(* IEC 61131-3 sources: fse/dataset/original (part 3) *)

(* ---- lb_claude_assisted_30195e188caf_0084.st ---- *)
TYPE
  LOGLEVEL : (CRITICAL, WARNING, INFO, DEBUG) := INFO;
END_TYPE

FUNCTION_BLOCK LOGGER
  VAR_INPUT
    TRIG : BOOL;
    MSG : STRING;
    LEVEL : LOGLEVEL := INFO;
  END_VAR
  VAR
    TRIG0 : BOOL;
  END_VAR

  IF TRIG AND NOT TRIG0 THEN
  {{
   LogMessage(GetFbVar(LEVEL),(char*)GetFbVar(MSG, .body),GetFbVar(MSG, .len));
  }}
  END_IF;
  TRIG0:=TRIG;
END_FUNCTION_BLOCK

FUNCTION_BLOCK python_eval
  VAR_INPUT
    TRIG : BOOL;
    CODE : STRING;
  END_VAR
  VAR_OUTPUT
    ACK : BOOL;
    RESULT : STRING;
  END_VAR
  VAR
    STATE : DWORD;
    BUFFER : STRING;
    PREBUFFER : STRING;
    TRIGM1 : BOOL;
    TRIGGED : BOOL;
  END_VAR

  {extern void __PythonEvalFB(int, PYTHON_EVAL*);__PythonEvalFB(0, data__);}
END_FUNCTION_BLOCK

FUNCTION_BLOCK python_poll
  VAR_INPUT
    TRIG : BOOL;
    CODE : STRING;
  END_VAR
  VAR_OUTPUT
    ACK : BOOL;
    RESULT : STRING;
  END_VAR
  VAR
    STATE : DWORD;
    BUFFER : STRING;
    PREBUFFER : STRING;
    TRIGM1 : BOOL;
    TRIGGED : BOOL;
  END_VAR

  {extern void __PythonEvalFB(int, PYTHON_EVAL*);__PythonEvalFB(1,(PYTHON_EVAL*)(void*)data__);}
END_FUNCTION_BLOCK

FUNCTION_BLOCK python_gear
  VAR_INPUT
    N : UINT;
    TRIG : BOOL;
    CODE : STRING;
  END_VAR
  VAR_OUTPUT
    ACK : BOOL;
    RESULT : STRING;
  END_VAR
  VAR
    py_eval : python_eval;
    COUNTER : UINT;
    _TMP_ADD10_OUT : UINT;
    _TMP_EQ13_OUT : BOOL;
    _TMP_SEL15_OUT : UINT;
    _TMP_AND7_OUT : BOOL;
  END_VAR

  _TMP_ADD10_OUT := ADD(COUNTER, 1);
  _TMP_EQ13_OUT := EQ(N, _TMP_ADD10_OUT);
  _TMP_SEL15_OUT := SEL(_TMP_EQ13_OUT, _TMP_ADD10_OUT, 0);
  COUNTER := _TMP_SEL15_OUT;
  _TMP_AND7_OUT := AND(_TMP_EQ13_OUT, TRIG);
  py_eval(TRIG := _TMP_AND7_OUT, CODE := CODE);
  ACK := py_eval.ACK;
  RESULT := py_eval.RESULT;
END_FUNCTION_BLOCK

PROGRAM plc2
  VAR
    ColorSensor_RED : INT;
    ColorSensor_GREEN : INT;
    ColorSensor_BLUE : INT;
    RangeSensor : REAL := 100.0;
    Pump : BOOL := FALSE;
    Doser_RED : BOOL := FALSE;
    Doser_BLUE : BOOL := FALSE;
  END_VAR
  VAR
    settleTime : TIME := TIME#5s;
    doseTime : TIME := TIME#1s;
    shutDown : BOOL := FALSE;
    treatmentComplete : BOOL := FALSE;
  END_VAR
  VAR
    stage : INT := 0;
    desiredDistanceFill : REAL := 60.0;
  END_VAR
  VAR
    minRed : INT := 20;
    doseTimer : TON;
    settleTimer : TON;
  END_VAR

  CASE stage OF
      0:  (*Filling stage: it will fill up to a certain amount that corresponds to a certain distance*)

          IF RangeSensor > desiredDistanceFill THEN
            Pump := TRUE;
          ELSE
            Pump := FALSE;
            stage := 1;
          END_IF;

     1:  (*Treatment stage*)

          IF ColorSensor_RED < minRed THEN (*Ensure minimum red value is inserted*)
            stage := 2;
            Doser_RED := TRUE;
            doseTimer(IN:= NOT doseTimer.Q, PT:= doseTime);

          ELSIF ColorSensor_RED > ColorSensor_BLUE  THEN (*Ensure blue quantity is > Red *)

              stage := 3;
              Doser_BLUE := TRUE;
              doseTimer(IN:= NOT doseTimer.Q, PT:= doseTime);

          ELSE  (*Treatment complete*)

            stage := 5;

          END_IF;

      2:  (*Red Dosing Stage*)

          IF doseTimer.Q THEN
            Doser_RED := FALSE;
            stage := 4;
            doseTimer(IN:= FALSE);
            settleTimer(IN:= NOT settleTimer.Q, PT:= settleTime); (*let the dose settle*)
          END_IF;

      3: (* Blue Dosing Stage*)

          IF doseTimer.Q THEN
            Doser_BLUE := FALSE;
            stage := 4;
            doseTimer(IN:= FALSE);
            settleTimer(IN:= NOT settleTimer.Q, PT:= settleTime); (*let the dose settle*)
          END_IF;

      4: (*Settling Stage for Dosage*)

          IF settleTimer.Q THEN
          stage := 1;
          settleTimer(IN:=FALSE);
          END_IF;

      5: (*Treatment Complete*)

        treatmentComplete := TRUE;

  END_CASE;
END_PROGRAM

CONFIGURATION Config0

  RESOURCE Res0 ON PLC
    TASK task0(INTERVAL := T#200ms,PRIORITY := 0);
    PROGRAM instance0 WITH task0 : plc2;
  END_RESOURCE
END_CONFIGURATION

(* ---- lb_claude_assisted_30f898e237c2_0134.st ---- *)
FUNCTION_BLOCK T_PLC_MS_block
	VAR_OUTPUT
		T_PLC_MS :	UDINT;
	END_VAR

	VAR_EXTERNAL
		PLC_TICKS_PER_SEC :	INT;
		PLC_SYS_TICK_CNT :	DINT;
	END_VAR

	VAR
		debug :	BOOL;(*Debug-Mode ON / OFF*)
		N :	INT;(*Debug-Faktor*)
		Offset :	UDINT;(*Debug-Offset*)
		temp :	DWORD := DWORD#1;(*Debug-Offset*)
		mode :	BOOL;(*modus*)
		faktor :	UDINT;(*Systemtakt-Faktor*)
		init :	BOOL;
		v_plc_ticks_per_sec :	UDINT;
		base :	UDINT := UDINT#1000;
	END_VAR

	IF init = FALSE THEN
		v_plc_ticks_per_sec := INT_TO_UDINT(PLC_TICKS_PER_SEC);
		IF v_plc_ticks_per_sec = UDINT#1024 THEN
			faktor := UDINT#1;
			mode := FALSE;
		ELSIF v_plc_ticks_per_sec > UDINT#0 THEN
			IF v_plc_ticks_per_sec <= base THEN
				faktor := base / v_plc_ticks_per_sec;
				mode := FALSE;
			ELSE
				faktor := v_plc_ticks_per_sec / base;
				mode := TRUE;
			END_IF;
		ELSE
			faktor := UDINT#1;
		END_IF;
		init := TRUE;
	END_IF;

	IF mode THEN
		T_PLC_MS := DINT_TO_UDINT(PLC_SYS_TICK_CNT) / faktor;
	ELSE
		T_PLC_MS := DINT_TO_UDINT(PLC_SYS_TICK_CNT) * faktor;
	END_IF;

	IF debug THEN
		T_PLC_MS := (DWORD_TO_UDINT(SHL(UDINT_TO_DWORD(T_PLC_MS),N) OR SHL(temp,N)) - UDINT#1) + Offset;
	END_IF;
END_FUNCTION_BLOCK

FUNCTION_BLOCK INTEGRATE

	VAR_INPUT
		E :	BOOL := TRUE;
		X :	REAL;
		K :	REAL := 1.0;
	END_VAR

	VAR_IN_OUT
		Y :	REAL;
	END_VAR

	VAR
		X_last :	REAL;
		init :	BOOL;
		T_PLC_MS :	T_PLC_MS_block;
		last :	UDINT;
		tx :	UDINT;
	END_VAR

	T_PLC_MS();
	tx:= T_PLC_MS.T_PLC_MS;

	IF NOT init THEN
		init := TRUE;
		X_last := X;
	ELSIF E THEN
		Y := (X + X_LAST) * 0.5E-3 * UDINT_TO_REAL(tx-last) * K + Y;
		X_last := X;
	END_IF;
	last := tx;

END_FUNCTION_BLOCK

FUNCTION_BLOCK FT_INT_Block

	VAR_INPUT
		IN :	REAL;
		K :	REAL := 1.0;
		RUN :	BOOL := TRUE;
		RST :	BOOL;
		OUT_MIN :	REAL := REAL#-1.0E-37;
		OUT_MAX :	REAL := REAL#1.0E37;
	END_VAR

	VAR_OUTPUT
		OUT :	REAL;
		LIM :	BOOL;
	END_VAR

	VAR
		INTEG :	INTEGRATE;
	END_VAR

	IF rst THEN
		out := 0.0;
	ELSE
		integ(X := IN, E := RUN, K := K, Y := out);
		out := integ.Y;
	END_IF;

	(* limit the outputs *)
	IF out >= OUT_MAX THEN
		out := out_max;
		LIM := TRUE;
	ELSIF out <= out_min THEN
		out := out_min;
		lim := TRUE;
	ELSE
		lim := FALSE;
	END_IF;

END_FUNCTION_BLOCK

FUNCTION_BLOCK FT_PIW

	VAR_INPUT
		IN :	REAL;
		KP :	REAL := 1.0;
		KI :	REAL := 1.0;
		LIM_L :	REAL := -1.0E38;
		LIM_H :	REAL := 1.0E38;
		RST :	BOOL := FALSE;
	END_VAR

	VAR_OUTPUT
		Y :	REAL;
		LIM :	BOOL;
	END_VAR

	VAR
		integ :	FT_INT_Block;
	END_VAR

	integ(IN := IN, K := KI, RUN := NOT LIM, RST := RST);

	(* set output value *)
	Y := KP * IN + integ.Out;

	(* check for limits *)
	IF Y < LIM_L THEN
		Y := LIM_L;
		LIM := TRUE;
	ELSIF Y > LIM_H THEN
		Y := LIM_H;
		LIM := TRUE;
	ELSE
		LIM := FALSE;
	END_IF;

END_FUNCTION_BLOCK

PROGRAM program0
	VAR
		IN :	REAL;
		KP :	REAL := 1.0;
		KI :	REAL := 1.0;
		LIM_L :	REAL := -1.0E38;
		LIM_H :	REAL := 1.0E38;
		RST :	BOOL := FALSE;

		Y :	REAL;
		LIM :	BOOL;

		func_block : FT_PIW;
	END_VAR
	func_block.IN := IN;
	func_block.KP := KP;
	func_block.KI := KI;
	func_block.LIM_L := LIM_L;
	func_block.LIM_H := LIM_H;
	func_block.RST := RST;
	func_block();
	Y := func_block.Y;
	LIM := func_block.LIM;
END_PROGRAM

CONFIGURATION Config0

	VAR_GLOBAL
		PLC_TICKS_PER_SEC :	INT;
		PLC_SYS_TICK_CNT :	DINT;
	END_VAR

	RESOURCE Res0 ON PLC
		TASK task0(INTERVAL := T#20ms,PRIORITY := 0);
		PROGRAM instance0 WITH task0 : program0;
	END_RESOURCE

END_CONFIGURATION

(* ---- lb_claude_assisted_33ab4d28fcd8_0080.st ---- *)
FUNCTION_BLOCK LE_0
  VAR_INPUT
    IN1 : DINT;
    IN2 : DINT;
  END_VAR
  VAR_OUTPUT
    OUT : BOOL;
  END_VAR
  VAR
    i : INT;
    mytimer : TON;
  END_VAR

  OUT:=FALSE;
  IF IN1<=IN2 then
    OUT:=TRUE;
  END_IF;
  mytimer(IN := TRUE, PT := t#8000ms);
  i:=0;
  IF mytimer.Q = TRUE then
     WHILE i<4 do
      OUT:=TRUE;
    End_WHILE;
  End_IF;
END_FUNCTION_BLOCK

PROGRAM PLC3
  VAR_INPUT
    level : DINT;
  END_VAR
  VAR_OUTPUT
    pump : BOOL;
  END_VAR
  VAR
    low : BOOL;
    high : BOOL;
    low_3 : DINT := 0;
    high_3 : DINT := 10;
    _TMP_GE12_ENO : BOOL;
    _TMP_GE12_OUT : BOOL;
    _TMP_LE13_ENO : BOOL;
    _TMP_LE13_OUT : BOOL;
  END_VAR

  _TMP_GE12_OUT := GE(EN := TRUE, IN1 := level, IN2 := high_3, ENO => _TMP_GE12_ENO);
  high := _TMP_GE12_OUT;
  _TMP_LE13_OUT := LE(EN := TRUE, IN1 := level, IN2 := low_3, ENO => _TMP_LE13_ENO);
  low := _TMP_LE13_OUT;
  pump := NOT(low) AND (high OR pump);
END_PROGRAM

PROGRAM PLC2
  VAR_INPUT
    level : DINT;
  END_VAR
  VAR_OUTPUT
    request : BOOL;
  END_VAR
  VAR
    open_req : BOOL;
    close_req : BOOL;
    low_2 : DINT := 10;
    high_2 : DINT := 20;
    LE_00 : LE_0;
    _TMP_GE11_ENO : BOOL;
    _TMP_GE11_OUT : BOOL;
  END_VAR

  _TMP_GE11_OUT := GE(EN := TRUE, IN1 := level, IN2 := high_2, ENO => _TMP_GE11_ENO);
  close_req := _TMP_GE11_OUT;
  LE_00(EN := TRUE, IN1 := level, IN2 := low_2);
  open_req := LE_00.OUT;
  request := NOT(close_req) AND (open_req OR request);
END_PROGRAM

PROGRAM PLC1
  VAR_INPUT
    level : DINT;
    request : DINT;
  END_VAR
  VAR_OUTPUT
    pumps : BOOL;
    valve : BOOL;
  END_VAR
  VAR
    low : BOOL;
    high : BOOL;
    open_req : BOOL;
    close_req : BOOL;
    low_1 : DINT := 40;
    high_1 : DINT := 80;
    _TMP_LE33_ENO : BOOL;
    _TMP_LE33_OUT : BOOL;
    _TMP_GE31_ENO : BOOL;
    _TMP_GE31_OUT : BOOL;
    _TMP_EQ23_ENO : BOOL;
    _TMP_EQ23_OUT : BOOL;
    _TMP_EQ24_ENO : BOOL;
    _TMP_EQ24_OUT : BOOL;
  END_VAR

  _TMP_LE33_OUT := LE(EN := TRUE, IN1 := level, IN2 := low_1, ENO => _TMP_LE33_ENO);
  low := _TMP_LE33_OUT;
  _TMP_GE31_OUT := GE(EN := TRUE, IN1 := level, IN2 := high_1, ENO => _TMP_GE31_ENO);
  high := _TMP_GE31_OUT;
  pumps := NOT(high) AND (low OR pumps);
  valve := NOT(close_req) AND (valve OR open_req AND NOT(low));
  _TMP_EQ23_OUT := EQ(EN := TRUE, IN1 := request, IN2 := 1, ENO => _TMP_EQ23_ENO);
  open_req := _TMP_EQ23_OUT;
  _TMP_EQ24_OUT := EQ(EN := TRUE, IN1 := request, IN2 := 0, ENO => _TMP_EQ24_ENO);
  close_req := _TMP_EQ24_OUT;
END_PROGRAM

CONFIGURATION Config0

  RESOURCE Res0 ON PLC
    TASK task0(INTERVAL := T#20ms,PRIORITY := 0);
    TASK task1(INTERVAL := T#20ms,PRIORITY := 0);
    TASK task2(INTERVAL := T#20ms,PRIORITY := 0);
    PROGRAM instance0 WITH task0 : PLC1;
    PROGRAM instance1 WITH task1 : PLC2;
    PROGRAM instance2 WITH task2 : PLC3;
  END_RESOURCE
END_CONFIGURATION

(* ---- lb_claude_assisted_33b79055e2cc_0056.st ---- *)
FUNCTION_BLOCK T_PLC_MS_block

	VAR_OUTPUT
		T_PLC_MS :	UDINT;
	END_VAR

	VAR_EXTERNAL
		PLC_TICKS_PER_SEC :	INT;
		PLC_SYS_TICK_CNT :	DINT;
	END_VAR

	VAR
		debug :	BOOL;(*Debug-Mode ON / OFF*)
		N :	INT;(*Debug-Faktor*)
		Offset :	UDINT;(*Debug-Offset*)
		temp :	DWORD := DWORD#1;(*Debug-Offset*)
		mode :	BOOL;(*modus*)
		faktor :	UDINT;(*Systemtakt-Faktor*)
		init :	BOOL;
		v_plc_ticks_per_sec :	UDINT;
		base :	UDINT := UDINT#1000;
	END_VAR

	IF init = FALSE THEN
		v_plc_ticks_per_sec := INT_TO_UDINT(PLC_TICKS_PER_SEC);
		IF v_plc_ticks_per_sec = UDINT#1024 THEN
			faktor := UDINT#1;
			mode := FALSE;
		ELSIF v_plc_ticks_per_sec > UDINT#0 THEN
			IF v_plc_ticks_per_sec <= base THEN
				faktor := base / v_plc_ticks_per_sec;
				mode := FALSE;
			ELSE
				faktor := v_plc_ticks_per_sec / base;
				mode := TRUE;
			END_IF;
		ELSE
			faktor := UDINT#1;
		END_IF;
		init := TRUE;
	END_IF;

	IF mode THEN
		T_PLC_MS := DINT_TO_UDINT(PLC_SYS_TICK_CNT) / faktor;
	ELSE
		T_PLC_MS := DINT_TO_UDINT(PLC_SYS_TICK_CNT) * faktor;
	END_IF;

	IF debug THEN
		T_PLC_MS := (DWORD_TO_UDINT(SHL(UDINT_TO_DWORD(T_PLC_MS),N) OR SHL(temp,N)) - UDINT#1) + Offset;
	END_IF;

END_FUNCTION_BLOCK

PROGRAM program0

	VAR
		LocalOUT  : UDINT;
		func_block : T_PLC_MS_block;
  	END_VAR

	func_block();
	LocalOUT := func_block.T_PLC_MS;

END_PROGRAM

CONFIGURATION Config0

	VAR_GLOBAL
		PLC_TICKS_PER_SEC :	INT;
		PLC_SYS_TICK_CNT :	DINT;
	END_VAR

  	RESOURCE Res0 ON PLC
    	TASK task0(INTERVAL := T#20ms,PRIORITY := 0);
    	PROGRAM instance0 WITH task0 : program0;
  	END_RESOURCE

END_CONFIGURATION

(* ---- lb_claude_assisted_350444d9c29e_0021.st ---- *)
(*
This code implements a randomly grown symbolic expression:

xor(xor(!((!(((xor(xor(((!(IN45)) & (IN32 | IN40)) & ((IN23 | IN38) | (!(IN24))), xor(xor((IN15 | IN19) & IN39, !(IN4 & IN13)), (xor(xor(IN43, IN11), IN25)) & (IN25 | IN49))), IN19)) | (xor(xor(IN43 & ((IN16 & IN26) | (!(IN43))), IN24 | ((!(IN13)) | IN33)), xor(xor(IN32, (IN20 & IN40) | (IN18 | IN23)), (IN42 & IN39) & (!(IN6)))))) & (!(IN16 & (xor(xor(!(IN50 & IN37), IN25), IN4)))))) & (!(!(((!(xor(xor(IN29 | IN47, xor(xor(IN44, IN42), IN1)), IN48 & IN20))) & (xor(xor((!(IN19)) | (IN47 & IN15), !(xor(xor(IN3, IN39), IN10))), xor(xor(IN35, IN48), IN40 & IN6)))) | (xor(xor(IN2, IN12), !(IN1))))))), IN30 | ((((xor(xor(((xor(xor(IN20 & IN48, !(IN20)), xor(xor(IN21, IN15), IN38))) & ((!(IN47)) & (IN13 & IN31))) & IN25, (((!(IN17)) | (IN34 | IN40)) | IN35) | ((xor(xor(IN37 | IN35, IN11 | IN33), !(IN9))) & ((IN43 & IN14) & (!(IN26))))), (xor(xor(xor(xor(IN45 & IN37, !(IN12)), IN4 | IN33), xor(xor(IN40, IN6 | IN14), IN38)), xor(xor(IN47 & IN30, IN29), !(IN36)))) | ((!(IN17)) | (xor(xor(IN45 | IN20, IN46 & IN36), !(IN17)))))) & (IN31 | (!(((IN9 | IN39) | (IN1 | IN44)) | (!(IN39 | IN42)))))) & IN41) & (((xor(xor(!(IN41 & (xor(xor(IN26 | IN47, xor(xor(IN25, IN44), IN28)), !(IN22)))), IN30), !(!(IN7 | (xor(xor(IN15, IN18), IN35)))))) | IN43) & (((xor(xor((xor(xor(!(IN37), xor(xor(IN36, IN29), IN20)), IN45)) | (xor(xor(IN24, xor(xor(IN17, IN22), IN40)), IN33 & IN36)), xor(xor(IN9 & (xor(xor(IN8, IN7), IN1)), IN29 | (IN49 | IN38)), xor(xor(IN48 | IN37, xor(xor(IN40, IN21), IN27)), !(IN9)))), !((xor(xor(IN21, IN35), IN17)) | IN47))) | IN41) | (IN40 & ((!(xor(xor(IN14 | IN35, IN10), true & IN31))) & (xor(xor((!(IN11)) | (!(IN1)), IN28), xor(xor(IN12, IN14 | IN38), IN26 & IN23))))))))), false)

*)

FUNCTION_BLOCK F_CollectInput
  VAR_IN_OUT
      Data : ARRAY[1..50] OF BOOL;
  END_VAR
  VAR_INPUT
      TICK  : BOOL := 0;
      IN1   : BOOL := 0;
      IN2   : BOOL := 0;
      IN3   : BOOL := 0;
      IN4   : BOOL := 0;
      IN5   : BOOL := 0;
      RESET : BOOL := FALSE;
  END_VAR
  VAR_OUTPUT
      Finished : BOOL;
  END_VAR
  VAR
      j    : USINT := 1;
      tock : BOOL  := 0;
  END_VAR
  IF NOT RESET AND tock = NOT TICK THEN
      Data[j]   := IN1;
      Data[j+1] := IN2;
      Data[j+2] := IN3;
      Data[j+3] := IN4;
      Data[j+4] := IN5;
      j := j + 5;
      tock := TICK;
  ELSE
      j := 1;
      tock := 0;
  END_IF;
  Finished := (j > 50);
END_FUNCTION_BLOCK

PROGRAM Boiler
  VAR
    Data  : ARRAY[1..50] OF BOOL;
    Ready : BOOL;
    CollectInput : F_CollectInput;
  END_VAR
  VAR
    TICK     AT %IX1.0 : BOOL;
    IN1      AT %IX0.3 : BOOL;
    IN2      AT %IX0.4 : BOOL;
    IN3      AT %IX0.5 : BOOL;
    IN4      AT %IX0.6 : BOOL;
    IN5      AT %IX0.7 : BOOL;
    OutReady AT %QX0.0 : BOOL := FALSE;
    FeedNext AT %QX0.1 : BOOL := FALSE;
    Out      AT %QX0.2 : BOOL;
  END_VAR
  CollectInput(TICK:=TICK, IN1:=IN1, IN2:=IN2, IN3:=IN3, IN4:=IN4, IN5:=IN5);
  Ready := CollectInput.Finished;
  FeedNext := 1;
  IF Ready THEN
    Out := (((NOT ((NOT (((((((NOT Data[45]) AND (Data[32] OR Data[40])) AND ((Data[23] OR Data[38]) OR (NOT Data[24]))) XOR ((((Data[15] OR Data[19]) AND Data[39]) XOR (NOT (Data[4] AND Data[13]))) XOR (((Data[43] XOR Data[11]) XOR Data[25]) AND (Data[25] OR Data[49])))) XOR Data[19]) OR (((Data[43] AND ((Data[16] AND Data[26]) OR (NOT Data[43]))) XOR (Data[24] OR ((NOT Data[13]) OR Data[33]))) XOR ((Data[32] XOR ((Data[20] AND Data[40]) OR (Data[18] OR Data[23]))) XOR ((Data[42] AND Data[39]) AND (NOT Data[6]))))) AND (NOT (Data[16] AND (((NOT (Data[50] AND Data[37])) XOR Data[25]) XOR Data[4]))))) AND (NOT (NOT (((NOT (((Data[29] OR Data[47]) XOR ((Data[44] XOR Data[42]) XOR Data[1])) XOR (Data[48] AND Data[20]))) AND ((((NOT Data[19]) OR (Data[47] AND Data[15])) XOR (NOT ((Data[3] XOR Data[39]) XOR Data[10]))) XOR ((Data[35] XOR Data[48]) XOR (Data[40] AND Data[6])))) OR ((Data[2] XOR Data[12]) XOR (NOT Data[1]))))))) XOR (Data[30] OR ((((((((((Data[20] AND Data[48]) XOR (NOT Data[20])) XOR ((Data[21] XOR Data[15]) XOR Data[38])) AND ((NOT Data[47]) AND (Data[13] AND Data[31]))) AND Data[25]) XOR ((((NOT Data[17]) OR (Data[34] OR Data[40])) OR Data[35]) OR ((((Data[37] OR Data[35]) XOR (Data[11] OR Data[33])) XOR (NOT Data[9])) AND ((Data[43] AND Data[14]) AND (NOT Data[26]))))) XOR ((((((Data[45] AND Data[37]) XOR (NOT Data[12])) XOR (Data[4] OR Data[33])) XOR ((Data[40] XOR (Data[6] OR Data[14])) XOR Data[38])) XOR (((Data[47] AND Data[30]) XOR Data[29]) XOR (NOT Data[36]))) OR ((NOT Data[17]) OR (((Data[45] OR Data[20]) XOR (Data[46] AND Data[36])) XOR (NOT Data[17]))))) AND (Data[31] OR (NOT (((Data[9] OR Data[39]) OR (Data[1] OR Data[44])) OR (NOT (Data[39] OR Data[42])))))) AND Data[41]) AND (((((NOT (Data[41] AND (((Data[26] OR Data[47]) XOR ((Data[25] XOR Data[44]) XOR Data[28])) XOR (NOT Data[22])))) XOR Data[30]) XOR (NOT (NOT (Data[7] OR ((Data[15] XOR Data[18]) XOR Data[35]))))) OR Data[43]) AND ((((((((NOT Data[37]) XOR ((Data[36] XOR Data[29]) XOR Data[20])) XOR Data[45]) OR ((Data[24] XOR ((Data[17] XOR Data[22]) XOR Data[40])) XOR (Data[33] AND Data[36]))) XOR (((Data[9] AND ((Data[8] XOR Data[7]) XOR Data[1])) XOR (Data[29] OR (Data[49] OR Data[38]))) XOR (((Data[48] OR Data[37]) XOR ((Data[40] XOR Data[21]) XOR Data[27])) XOR (NOT Data[9])))) XOR (NOT (((Data[21] XOR Data[35]) XOR Data[17]) OR Data[47]))) OR Data[41]) OR (Data[40] AND ((NOT (((Data[14] OR Data[35]) XOR Data[10]) XOR (TRUE AND Data[31]))) AND ((((NOT Data[11]) OR (NOT Data[1])) XOR Data[28]) XOR ((Data[12] XOR (Data[14] OR Data[38])) XOR (Data[26] AND Data[23])))))))))) XOR FALSE);
    OutReady := 1;
    CollectInput(RESET:=TRUE);
  END_IF;
END_PROGRAM

CONFIGURATION Config0
  RESOURCE Res0 ON PLC
    TASK task0(INTERVAL := T#20ms,PRIORITY := 0);
    PROGRAM instance0 WITH task0 : Boiler;
  END_RESOURCE
END_CONFIGURATION

(* ---- lb_claude_assisted_3919578456ab_0001.st ---- *)
FUNCTION_BLOCK T_PLC_MS_block
	VAR_OUTPUT
		T_PLC_MS :	UDINT;
	END_VAR

	VAR
		PLC_TICKS_PER_SEC :	INT;
		PLC_SYS_TICK_CNT :	DINT;
	END_VAR

	VAR
		debug :	BOOL;(*Debug-Mode ON / OFF*)
		N :	INT;(*Debug-Faktor*)
		Offset :	UDINT;(*Debug-Offset*)
		temp :	DWORD := DWORD#1;(*Debug-Offset*)
		MODE :	BOOL;(*modus*)
		faktor :	UDINT;(*Systemtakt-Faktor*)
		init :	BOOL;
		v_plc_ticks_per_sec :	UDINT;
		base :	UDINT := UDINT#1000;
	END_VAR

	IF init = FALSE THEN
		v_plc_ticks_per_sec := INT_TO_UDINT(PLC_TICKS_PER_SEC);
		IF v_plc_ticks_per_sec = UDINT#1024 THEN
			faktor := UDINT#1;
			MODE := FALSE;
		ELSIF v_plc_ticks_per_sec > UDINT#0 THEN
			IF v_plc_ticks_per_sec <= base THEN
				faktor := base / v_plc_ticks_per_sec;
				MODE := FALSE;
			ELSE
				faktor := v_plc_ticks_per_sec / base;
				MODE := TRUE;
			END_IF;
		ELSE
			faktor := UDINT#1;
		END_IF;
		init := TRUE;
	END_IF;

	IF MODE THEN
		T_PLC_MS := DINT_TO_UDINT(PLC_SYS_TICK_CNT) / faktor;
	ELSE
		T_PLC_MS := DINT_TO_UDINT(PLC_SYS_TICK_CNT) * faktor;
	END_IF;

	IF debug THEN
		T_PLC_MS := (DWORD_TO_UDINT(SHL(UDINT_TO_DWORD(T_PLC_MS),N) OR SHL(temp,N)) - UDINT#1) + Offset;
	END_IF;

END_FUNCTION_BLOCK

FUNCTION_BLOCK CLK_PRG
	VAR_INPUT
		PT :	TIME := T#10ms;
	END_VAR

	VAR_OUTPUT
		Q :	BOOL;
	END_VAR

	VAR
		init :	BOOL := FALSE;
		last :	TIME;
		TX :	TIME;
		T_PLC_MS :	T_PLC_MS_block;
	END_VAR

	T_PLC_MS();
	TX:= UDINT_TO_TIME(T_PLC_MS.T_PLC_MS);

	IF NOT init THEN
		init := TRUE;
		last := SUB_TIME(TX, PT);
	END_IF;

	Q := SUB_TIME(TX, last) >= PT;
	IF Q THEN last := TX; END_IF;
END_FUNCTION_BLOCK

FUNCTION _REAL_TO_UDINT:UDINT
  VAR_INPUT
    X :	REAL;
  END_VAR

  IF REAL_TO_UDINT(0.5) = UDINT#1 THEN
    _REAL_TO_UDINT := REAL_TO_UDINT(X);
  ELSIF X > 0.0 THEN
    _REAL_TO_UDINT := REAL_TO_UDINT(X+0.5);
  ELSIF X < 0.0 THEN
    _REAL_TO_UDINT := REAL_TO_UDINT(X-0.5);
  ELSE
    _REAL_TO_UDINT := UDINT#0;
  END_IF;
END_FUNCTION

FUNCTION REAL_TO_TIME2:TIME
	VAR_INPUT
		IN :	REAL;
	END_VAR

	REAL_TO_TIME2 := DINT_TO_TIME(UDINT_TO_DINT(_REAL_TO_UDINT(IN)));
END_FUNCTION

FUNCTION_BLOCK TP_X
	VAR_INPUT
		IN :	BOOL;
		PT :	TIME;
	END_VAR

	VAR_OUTPUT
		Q :	BOOL;
		ET :	TIME;
	END_VAR

	VAR
		edge :	BOOL;
		START :	TIME;
		TX :	TIME;
		T_PLC_MS :	T_PLC_MS_block;
	END_VAR

	T_PLC_MS();
	TX := UDINT_TO_TIME(T_PLC_MS.T_PLC_MS);

	IF IN AND NOT edge THEN
		START := TX;
		Q := PT > t#0ms;
	ELSIF Q THEN
		ET := SUB_TIME (TX, START);
		IF ET >= PT THEN
			Q := FALSE;
			ET := t#0ms;
		END_IF;
	END_IF;
	edge := IN;

END_FUNCTION_BLOCK

FUNCTION_BLOCK PWM_DC
	VAR_INPUT
		F :	REAL;
		DC :	REAL;
	END_VAR

	VAR_OUTPUT
		Q :	BOOL;
	END_VAR

	VAR
		CLK :	CLK_PRG;
		pulse :	TP_X;
		tmp :	REAL;
	END_VAR

	IF F > 0.0 THEN
		tmp := 1000.0/F;
		CLK(PT := REAL_TO_TIME2(tmp));
		pulse(IN := CLK.Q, PT := REAL_TO_TIME2(tmp*DC));
		Q := pulse.Q;
	END_IF;
END_FUNCTION_BLOCK

FUNCTION_BLOCK CTRL_PWM
	VAR_INPUT
		CI :	REAL;
		MAN_IN :	REAL;
		MANUAL :	BOOL;
		F :	REAL;
	END_VAR

	VAR_OUTPUT
		Q :	BOOL;
	END_VAR

	VAR
		PW :	PWM_DC;
	END_VAR

	PW(F := F, DC := SEL(MANUAL,CI,MAN_IN));
	Q := PW.Q;
END_FUNCTION_BLOCK

PROGRAM program0
  VAR
	CI     :	REAL;
	MAN_IN :	REAL;
	MANUAL :	BOOL;
	F      :	REAL;

	Q :	BOOL;

	func_block : CTRL_PWM;
  END_VAR
	func_block.CI    :=CI    ;
	func_block.MAN_IN:=MAN_IN;
	func_block.MANUAL:=MANUAL;
	func_block.F     :=F     ;
	func_block();
	Q := func_block.Q;
END_PROGRAM

(* ---- lb_claude_assisted_3f90610631a6_0023.st ---- *)
(*
 *
 * File: sine_PLC.st
 *
 * IEC 61131-3 Structured Text (ST) code generated for subsystem "sine_PLC/Subsystem"
 *
 * Model name                      : sine_PLC
 * Model version                   : 1.0
 * Model creator                   : imkis
 * Model last modified by          : imkis
 * Model last modified on          : Wed Jun 03 14:36:07 2020
 * Model sample time               : 0s
 * Subsystem name                  : sine_PLC/Subsystem
 * Subsystem sample time           : 0.01s
 * Simulink PLC Coder version      : 3.2 (R2020a) 18-Nov-2019
 * ST code generated on            : Wed Jun 03 16:22:54 2020
 *
 * Target IDE selection            : Generic
 * Test Bench included             : No
 *
 *)
FUNCTION_BLOCK Subsystem
VAR_INPUT
    ssMethodType: SINT;
END_VAR
VAR_OUTPUT
    Current_command: INT;
END_VAR
VAR
    b_counter: DINT;
END_VAR
VAR_TEMP
    rtb_SineWave: LREAL;
END_VAR
CASE ssMethodType OF
    0:
        (* SystemInitialize for Atomic SubSystem: '<Root>/Subsystem' *)
        (* InitializeConditions for Sin: '<S1>/Sine Wave' *)
        b_counter := 0;
        (* End of SystemInitialize for SubSystem: '<Root>/Subsystem' *)
    1:
        (* Outputs for Atomic SubSystem: '<Root>/Subsystem' *)
        (* Sin: '<S1>/Sine Wave' *)
        rtb_SineWave := SIN(((DINT_TO_LREAL(b_counter) * 2.0) * 3.1415926535897931) / 100.0) * 500.0;
        (* Update for Sin: '<S1>/Sine Wave' *)
        b_counter := b_counter + 1;
        IF b_counter = 100 THEN
            b_counter := 0;
        END_IF;
        (* End of Update for Sin: '<S1>/Sine Wave' *)

        (* Outport: '<Root>/Current_command' incorporates:
         *  DataTypeConversion: '<S1>/Data Type Conversion' *)
        Current_command := DINT_TO_INT(TRUNC(rt_floord(u := rtb_SineWave)));
        (* End of Outputs for SubSystem: '<Root>/Subsystem' *)
END_CASE;
END_FUNCTION_BLOCK
FUNCTION rt_floord: LREAL
VAR_INPUT
    u: LREAL;
END_VAR
rt_floord := DINT_TO_LREAL(TRUNC(u));
IF u = rt_floord THEN
    rt_floord := u;
ELSIF u < 0.0 THEN
    rt_floord := rt_floord - 1.0;
END_IF;
END_FUNCTION

(* ---- lb_claude_assisted_421cef1b1973_0024.st ---- *)
FUNCTION T_PLC_US : UDINT
  VAR
    tx : UDINT;
  END_VAR
  VAR_INPUT
    debug : BOOL;
  END_VAR
  VAR
    N : INT := 0;
    offset : UDINT := 0;
    temp : DWORD := 1;
  END_VAR

  {extern unsigned long __tick;
  extern unsigned long long common_ticktime__;
  unsigned long long ticktime_ms = (common_ticktime__)/1000000;
  UDINT plc_time = (UDINT)(ticktime_ms * (unsigned long long)__tick);
  TX = plc_time}

  T_PLC_US := tx*1000;
  IF debug THEN
  	T_PLC_US := (DWORD_TO_UDINT(SHL(UDINT_TO_DWORD(T_PLC_US),N) OR SHL(temp,N))-1) + OFFSET;
  END_IF;

  (* Original Code:
  tx := TIME();
  T_PLC_US := TIME_TO_DWORD(Tx)*1000;
  IF debug THEN
  	T_PLC_US := (SHL(T_PLC_US,N) OR SHL(DWORD#1,N)-1) + OFFSET;
  END_IF;
  *)

  (* From OSCAT library, www.oscat.de

  this is a temporary T_PLC_US FB until OpenPLC gets it´s own time() functionality *)

  (* PLC_TIME and Global variables PLC_SCAN_CYCL and PLC_CYCL_TIME required *)
END_FUNCTION

FUNCTION_BLOCK FT_PIWL
  VAR_INPUT
    IN : REAL;
    KP : REAL := 1.0;
    KI : REAL := 1.0;
    LIM_L : REAL := -1.0E38;
    LIM_H : REAL := 1.0E38;
    RST : BOOL;
  END_VAR
  VAR_OUTPUT
    Y : REAL;
    LIM : BOOL;
  END_VAR
  VAR
    init : BOOL;
    tx : UDINT;
    tc : REAL;
    t_last : UDINT;
    in_last : REAL;
    i : REAL;
    p : REAL;
  END_VAR

  IF NOT init OR RST THEN
  	init := TRUE;
  	in_last := in;
  		t_last := T_PLC_US(en:=true);
  	i := 0.0;
  	tc := 0.0;
  ELSE
  	(* read last cycle time in Microseconds *)
  		tx := T_PLC_US(en:=true);
  	tc := UDINT_TO_REAL(tx - t_last);
  	t_last := tx;

  	(* calculate proportional part *)
  	p := KP * IN;

  	(* run integrator *)
  	i := (IN + in_last) * 5.0E-7 * KI * tc + i;
  	in_last := IN;

  	(* calculate output Y *)
  	Y := p + i;

  	(* check output for limits *)
  	IF Y >= LIM_H THEN
  		Y := LIM_H;
  		IF ki <> 0.0 THEN
  			i := LIM_H - p;
  		ELSE
  			i := 0.0;
  		END_IF;
  		LIM := TRUE;
  	ELSIF Y <= LIM_L THEN
  		Y := LIM_L;
  		IF ki <> 0.0 THEN
  			i := LIM_L - p;
  		ELSE
  			i := 0.0;
  		END_IF;
  		LIM := TRUE;
  	ELSE
  		LIM := FALSE;
  	END_IF;
  END_IF;

  (* From OSCAT Library, www.oscat.de *)
  (* T_PLC_US required *)
END_FUNCTION_BLOCK

FUNCTION_BLOCK FT_DERIV
  VAR_INPUT
    IN : REAL;
    K : REAL := 1.0;
    RUN : BOOL := TRUE;
  END_VAR
  VAR_OUTPUT
    OUT : REAL;
  END_VAR
  VAR
    old : REAL;
    tx : UDINT;
    last : UDINT;
    init : BOOL;
    tc : REAL;
  END_VAR

  tx:= T_PLC_US(en:=true);
  tc := UDINT_TO_REAL(tx - last);

  (* init on firsat startup *)
  IF NOT init THEN
  	init := TRUE;
  	old := in;
  ELSIF run AND tc > 0.0 THEN
  	out := (in - old) / tc * 1000000.0 * K;
  	old := in;
  ELSE
  	out := 0.0;
  END_IF;

  last := tx;

  (* From OSCAT Library, www.oscat.de *)
  (* T_PLC_US, required *)
END_FUNCTION_BLOCK

FUNCTION_BLOCK FT_PIDWL
  VAR_INPUT
    IN : REAL;
    KP : REAL := 1.0;
    TN : REAL := 1.0;
    TV : REAL := 1.0;
    LIM_L : REAL := -1.0E38;
    LIM_H : REAL := 1.0E38;
    RST : BOOL;
  END_VAR
  VAR_OUTPUT
    Y : REAL;
    LIM : BOOL;
  END_VAR
  VAR
    piwl : FT_PIWL;
    diff : FT_DERIV;
  END_VAR

  IF rst THEN
  	piwl(rst := TRUE);
  	piwl.RST := FALSE;
  ELSE
  	(* run PIWL controller first *)
  	(* we need to check if TN = 0 and do alternative calls *)
  	IF TN = 0.0 THEN
  		piwl(in := IN * KP, KP := 1.0, KI := 0.0, LIM_L := LIM_L, LIM_H := LIM_H);
  	ELSE
  		piwl(in := IN * KP, KP := 1.0, KI := 1.0 / TN, LIM_L := LIM_L, LIM_H := LIM_H);
  	END_IF;

  	(* run differentiator and add_to_output *)
  	diff(IN := IN, K := KP * TV);
  	Y := piwl.Y + diff.out;

  	(* limit the output *)
  	IF Y < LIM_L THEN
  		LIM := TRUE;
  		Y := LIM_L;
  	ELSIF Y > LIM_H THEN
  		LIM := TRUE;
  		Y := LIM_H;
  	ELSE
  		LIM := FALSE;
  	END_IF;
  END_IF;

  (* From OSCAT Library, www.oscat.de *)
  (* T_PLC_US, FT_DERIV required *)
END_FUNCTION_BLOCK

FUNCTION_BLOCK CTRL_OUT
  VAR_INPUT
    CI : REAL;
    OFFSET : REAL;
    MAN_IN : REAL;
    LIM_L : REAL;
    LIM_H : REAL;
    MANUAL : BOOL;
  END_VAR
  VAR_OUTPUT
    Y : REAL;
    LIM : BOOL;
  END_VAR

  Y := SEL(manual, CI, MAN_IN) + OFFSET;

  (* Limit the output *)
  IF Y >= LIM_H THEN
  	Y := LIM_H;
  	LIM := TRUE;
  ELSIF Y <= lim_L THEN
  	Y := LIM_L;
  	LIM := TRUE;
  ELSE
  	LIM := FALSE;
  END_IF;

  (* From OSCAT Library, www.oscat.de *)
END_FUNCTION_BLOCK

FUNCTION DEAD_ZONE : REAL
  VAR_INPUT
    X : REAL;
    L : REAL;
  END_VAR

  IF ABS(x) > L THEN
  	dead_zone := X;
  ELSE
  	DEAD_ZONE := 0.0;
  END_IF;

  (* From OSCAT Library, www.oscat.de *)
END_FUNCTION

FUNCTION CTRL_IN : REAL
  VAR_INPUT
    SET_POINT : REAL;
    ACTUAL : REAL;
    NOISE : REAL;
  END_VAR

  CTRL_IN := DEAD_ZONE(SET_POINT - ACTUAL, NOISE);

  (* From OSCAT Library, www.oscat.de *)
  (* DEAD_ZONE required *)
END_FUNCTION

FUNCTION_BLOCK CTRL_PID
  VAR_INPUT
    ACT : REAL;
    SET : REAL;
    SUP : REAL;
    OFS : REAL;
    M_I : REAL;
    MAN : BOOL;
    RST : BOOL := FALSE;
    KP : REAL := 1.0;
    TN : REAL := 1.0;
    TV : REAL := 1.0;
    LL : REAL := -1000.0;
    LH : REAL := 1000.0;
  END_VAR
  VAR_OUTPUT
    Y : REAL;
    DIFF : REAL;
    LIM : BOOL;
  END_VAR
  VAR
    _pid : FT_PIDWL;
    co : CTRL_OUT;
  END_VAR

  DIFF := CTRL_IN(SET, ACT, SUP);
  _pid(in := DIFF, kp := KP, tn := TN, tv := TV, lim_l := LL, lim_h := LH, rst := RST);
  co(ci := _pid.Y, OFFSET := OFS, man_in := M_I, lim_l := LL, lim_h := LH, manual := MAN);
  Y := co.Y;
  LIM := co.LIM;

  (* From OSCAT Library, www.oscat.de *)
  (* CTRL_IN, FT_PIDWL, CTRL_out reauired *)
END_FUNCTION_BLOCK

FUNCTION_BLOCK PID_Controller
  VAR_INPUT
    ACT : REAL;
    SET : REAL;
  END_VAR
  VAR
    ctrl_pid1 : CTRL_PID;
    ctrl_out1 : CTRL_OUT;
  END_VAR
  VAR_OUTPUT
    Y : REAL;
    DIFF : REAL;
    LIM : BOOL;
  END_VAR

  ctrl_pid1(ACT := ACT,
            SET := SET,
            SUP := 0.0,
            OFS := 0.0,
            M_I := 0.0,
            MAN := FALSE,
            RST := FALSE,
            KP := 1.0,
            TN := 1.0,
            TV := 1.0,
            LL := -100.0,
            LH := 100.0);
  Y := ctrl_pid1.Y;

  (*

  ctrl_out1(CI := ctrl_pid1.Y,
            MAN_IN := 0.0,
            MANUAL := FALSE,
            LIM_L := -100.0,
            LIM_H := 100.0);

  Y := ctrl_out1.Y;
  DIFF := ctrl_pid1.DIFF;
  LIM := ctrl_pid1.LIM;
  *)

END_FUNCTION_BLOCK

FUNCTION_BLOCK AMMONIUM_NITRATE_TEMP_CONTROL
  VAR_INPUT
    temp_actual : REAL;
    manual_mode : BOOL;
    manual_input : REAL;
  END_VAR
  VAR_OUTPUT
    control_output : REAL;
  END_VAR
  VAR
    set_point : REAL := 180.0;
    kp : REAL := 50.0;
    ki : REAL := 1.2;
    kd : REAL := 10.0;
    lower_limit : REAL := -100.0;
    upper_limit : REAL := 100.0;
    pidcontroller : CTRL_PID;
    timer : TON;
    timer_done : BOOL;
  END_VAR

  timer(IN:=NOT manual_mode, PT:=T#10S);
  timer_done := timer.Q;

  IF timer_done THEN
      pidcontroller(ACT:=temp_actual,
                     SET:=set_point,
                     KP:=kp,
                     TN:=kp/ki,
                     TV:=kd/kp,
                     LL:=lower_limit,
                     LH:=upper_limit,
                     MAN:=manual_mode,
                     M_I:=manual_input,
                     RST:=FALSE);
      control_output := pidcontroller.Y;
  ELSE
      control_output := 0.0;
  END_IF;
END_FUNCTION_BLOCK

PROGRAM program0
  VAR
    myACT : REAL := 0.1;
    mySET : REAL := 1.0;
    myPIDController : PID_Controller;
    myPID : AMMONIUM_NITRATE_TEMP_CONTROL;
  END_VAR

  (*
  myPIDController(ACT := myACT, SET := mySET);
  *)

  myPID(temp_actual := myAct,
        manual_mode := FALSE,
        manual_input := 0.0);

  IF myACT < mySET THEN
    myACT := myACT + 0.01;
  ELSIF myACT > mySET THEN
    myACT := myACT - 0.01;
  END_IF;

END_PROGRAM

CONFIGURATION Config0

  RESOURCE Res0 ON PLC
    TASK task0(INTERVAL := T#100ms,PRIORITY := 0);
    PROGRAM instance0 WITH task0 : program0;
  END_RESOURCE
END_CONFIGURATION

(* ---- lb_claude_assisted_4378e99e8c95_0034.st ---- *)
(*
This code implements a randomly grown symbolic expression:

!(!(xor(xor(IN7 | ((((!(xor(xor(IN46, IN6 & IN48), IN36 | IN35))) | (!((xor(xor(IN26, IN22), IN45)) | (IN5 | true)))) | (!(((IN23 & IN25) & IN7) | (xor(xor(xor(xor(IN6, IN4), true), xor(xor(IN2, IN20), IN9)), xor(xor(IN4, IN11), IN36)))))) & (!(IN23))), IN8), ((!((((IN36 & IN24) | (IN45 | IN45)) | ((!(IN8)) | (!(IN23)))) & ((xor(xor(xor(xor(IN41, IN42), IN5), xor(xor(IN5, IN3), IN41)), xor(xor(IN20, IN39), true))) & (xor(xor(!(IN12), IN47 & false), IN14 & IN23))))) | (xor(xor((!(IN3)) & (((xor(xor(IN24, IN43), IN28)) | (!(IN10))) & (!(IN22 | IN28))), IN16), (xor(xor(IN1, IN1), (IN16 & true) | (IN40 | IN50))) & (!(IN39 & (IN8 & IN8)))))) | IN3)))

*)

FUNCTION_BLOCK F_CollectInput
  VAR_IN_OUT
      Data : ARRAY[1..50] OF BOOL;
  END_VAR
  VAR_INPUT
      TICK  : BOOL := 0;
      IN1   : BOOL := 0;
      IN2   : BOOL := 0;
      IN3   : BOOL := 0;
      IN4   : BOOL := 0;
      IN5   : BOOL := 0;
      RESET : BOOL := FALSE;
  END_VAR
  VAR_OUTPUT
      Finished : BOOL;
  END_VAR
  VAR
      j    : USINT := 1;
      tock : BOOL  := 0;
  END_VAR
  IF NOT RESET AND tock = NOT TICK THEN
      Data[j]   := IN1;
      Data[j+1] := IN2;
      Data[j+2] := IN3;
      Data[j+3] := IN4;
      Data[j+4] := IN5;
      j := j + 5;
      tock := TICK;
  ELSE
      j := 1;
      tock := 0;
  END_IF;
  Finished := (j > 50);
END_FUNCTION_BLOCK

PROGRAM Boiler
  VAR
    Data  : ARRAY[1..50] OF BOOL;
    Ready : BOOL;
    CollectInput : F_CollectInput;
  END_VAR
  VAR
    TICK     AT %IX1.0 : BOOL;
    IN1      AT %IX0.3 : BOOL;
    IN2      AT %IX0.4 : BOOL;
    IN3      AT %IX0.5 : BOOL;
    IN4      AT %IX0.6 : BOOL;
    IN5      AT %IX0.7 : BOOL;
    OutReady AT %QX0.0 : BOOL := FALSE;
    FeedNext AT %QX0.1 : BOOL := FALSE;
    Out      AT %QX0.2 : BOOL;
  END_VAR
  CollectInput(TICK:=TICK, IN1:=IN1, IN2:=IN2, IN3:=IN3, IN4:=IN4, IN5:=IN5);
  Ready := CollectInput.Finished;
  FeedNext := 1;
  IF Ready THEN
    Out := (NOT (NOT (((Data[7] OR ((((NOT ((Data[46] XOR (Data[6] AND Data[48])) XOR (Data[36] OR Data[35]))) OR (NOT (((Data[26] XOR Data[22]) XOR Data[45]) OR (Data[5] OR TRUE)))) OR (NOT (((Data[23] AND Data[25]) AND Data[7]) OR ((((Data[6] XOR Data[4]) XOR TRUE) XOR ((Data[2] XOR Data[20]) XOR Data[9])) XOR ((Data[4] XOR Data[11]) XOR Data[36]))))) AND (NOT Data[23]))) XOR Data[8]) XOR (((NOT ((((Data[36] AND Data[24]) OR (Data[45] OR Data[45])) OR ((NOT Data[8]) OR (NOT Data[23]))) AND (((((Data[41] XOR Data[42]) XOR Data[5]) XOR ((Data[5] XOR Data[3]) XOR Data[41])) XOR ((Data[20] XOR Data[39]) XOR TRUE)) AND (((NOT Data[12]) XOR (Data[47] AND FALSE)) XOR (Data[14] AND Data[23]))))) OR ((((NOT Data[3]) AND ((((Data[24] XOR Data[43]) XOR Data[28]) OR (NOT Data[10])) AND (NOT (Data[22] OR Data[28])))) XOR Data[16]) XOR (((Data[1] XOR Data[1]) XOR ((Data[16] AND TRUE) OR (Data[40] OR Data[50]))) AND (NOT (Data[39] AND (Data[8] AND Data[8])))))) OR Data[3]))));
    OutReady := 1;
    CollectInput(RESET:=TRUE);
  END_IF;
END_PROGRAM

CONFIGURATION Config0
  RESOURCE Res0 ON PLC
    TASK task0(INTERVAL := T#20ms,PRIORITY := 0);
    PROGRAM instance0 WITH task0 : Boiler;
  END_RESOURCE
END_CONFIGURATION

(* ---- lb_claude_assisted_473197f4a314_0062.st ---- *)
(*
This code implements a randomly grown symbolic expression:

IN38 | IN6

*)

FUNCTION_BLOCK F_CollectInput
  VAR_IN_OUT
      Data : ARRAY[1..50] OF BOOL;
  END_VAR
  VAR_INPUT
      TICK  : BOOL := 0;
      IN1   : BOOL := 0;
      IN2   : BOOL := 0;
      IN3   : BOOL := 0;
      IN4   : BOOL := 0;
      IN5   : BOOL := 0;
      RESET : BOOL := FALSE;
  END_VAR
  VAR_OUTPUT
      Finished : BOOL;
  END_VAR
  VAR
      j    : USINT := 1;
      tock : BOOL  := 0;
  END_VAR
  IF NOT RESET AND tock = NOT TICK THEN
      Data[j]   := IN1;
      Data[j+1] := IN2;
      Data[j+2] := IN3;
      Data[j+3] := IN4;
      Data[j+4] := IN5;
      j := j + 5;
      tock := TICK;
  ELSE
      j := 1;
      tock := 0;
  END_IF;
  Finished := (j > 50);
END_FUNCTION_BLOCK

PROGRAM Boiler
  VAR
    Data  : ARRAY[1..50] OF BOOL;
    Ready : BOOL;
    CollectInput : F_CollectInput;
  END_VAR
  VAR
    TICK     AT %IX1.0 : BOOL;
    IN1      AT %IX0.3 : BOOL;
    IN2      AT %IX0.4 : BOOL;
    IN3      AT %IX0.5 : BOOL;
    IN4      AT %IX0.6 : BOOL;
    IN5      AT %IX0.7 : BOOL;
    OutReady AT %QX0.0 : BOOL := FALSE;
    FeedNext AT %QX0.1 : BOOL := FALSE;
    Out      AT %QX0.2 : BOOL;
  END_VAR
  CollectInput(TICK:=TICK, IN1:=IN1, IN2:=IN2, IN3:=IN3, IN4:=IN4, IN5:=IN5);
  Ready := CollectInput.Finished;
  FeedNext := 1;
  IF Ready THEN
    Out := (Data[38] OR Data[6]);
    OutReady := 1;
    CollectInput(RESET:=TRUE);
  END_IF;
END_PROGRAM

CONFIGURATION Config0
  RESOURCE Res0 ON PLC
    TASK task0(INTERVAL := T#20ms,PRIORITY := 0);
    PROGRAM instance0 WITH task0 : Boiler;
  END_RESOURCE
END_CONFIGURATION

(* ---- lb_claude_assisted_4cdbe01cfa0d_0077.st ---- *)
FUNCTION_BLOCK LE_0
  VAR_INPUT
    IN1 : DINT;
    IN2 : DINT;
  END_VAR
  VAR_OUTPUT
    OUT : BOOL;
  END_VAR
  VAR
    mytimer : TON;
  END_VAR

  OUT:=FALSE;
  IF IN1<=IN2 then
    OUT:=TRUE;
  END_IF;
  mytimer(IN := TRUE, PT := t#8000ms);

  IF mytimer.Q = TRUE then

      OUT:=TRUE;

  End_IF;
END_FUNCTION_BLOCK

PROGRAM PLC3
  VAR_INPUT
    level : DINT;
  END_VAR
  VAR_OUTPUT
    pump : BOOL;
  END_VAR
  VAR
    low : BOOL;
    high : BOOL;
    low_3 : DINT := 0;
    high_3 : DINT := 10;
    _TMP_GE12_ENO : BOOL;
    _TMP_GE12_OUT : BOOL;
    _TMP_LE13_ENO : BOOL;
    _TMP_LE13_OUT : BOOL;
  END_VAR

  _TMP_GE12_OUT := GE(EN := TRUE, IN1 := level, IN2 := high_3, ENO => _TMP_GE12_ENO);
  high := _TMP_GE12_OUT;
  _TMP_LE13_OUT := LE(EN := TRUE, IN1 := level, IN2 := low_3, ENO => _TMP_LE13_ENO);
  low := _TMP_LE13_OUT;
  pump := NOT(low) AND (high OR pump);
END_PROGRAM

PROGRAM PLC2
  VAR_INPUT
    level : DINT;
  END_VAR
  VAR_OUTPUT
    request : BOOL;
  END_VAR
  VAR
    open_req : BOOL;
    close_req : BOOL;
    low_2 : DINT := 10;
    high_2 : DINT := 20;
    LE_00 : LE_0;
    _TMP_GE11_ENO : BOOL;
    _TMP_GE11_OUT : BOOL;
  END_VAR

  LE_00(EN := TRUE, IN1 := level, IN2 := low_2);
  open_req := LE_00.OUT;
  _TMP_GE11_OUT := GE(EN := TRUE, IN1 := level, IN2 := high_2, ENO => _TMP_GE11_ENO);
  close_req := _TMP_GE11_OUT;
  request := NOT(close_req) AND (open_req OR request);
END_PROGRAM

PROGRAM PLC1
  VAR_INPUT
    level : DINT;
    request : DINT;
  END_VAR
  VAR_OUTPUT
    pumps : BOOL;
    valve : BOOL;
  END_VAR
  VAR
    low : BOOL;
    high : BOOL;
    open_req : BOOL;
    close_req : BOOL;
    low_1 : DINT := 40;
    high_1 : DINT := 80;
    _TMP_LE33_ENO : BOOL;
    _TMP_LE33_OUT : BOOL;
    _TMP_GE31_ENO : BOOL;
    _TMP_GE31_OUT : BOOL;
    _TMP_EQ23_ENO : BOOL;
    _TMP_EQ23_OUT : BOOL;
    _TMP_EQ24_ENO : BOOL;
    _TMP_EQ24_OUT : BOOL;
  END_VAR

  _TMP_LE33_OUT := LE(EN := TRUE, IN1 := level, IN2 := low_1, ENO => _TMP_LE33_ENO);
  low := _TMP_LE33_OUT;
  _TMP_GE31_OUT := GE(EN := TRUE, IN1 := level, IN2 := high_1, ENO => _TMP_GE31_ENO);
  high := _TMP_GE31_OUT;
  pumps := NOT(high) AND (low OR pumps);
  valve := NOT(close_req) AND (valve OR open_req AND NOT(low));
  _TMP_EQ23_OUT := EQ(EN := TRUE, IN1 := request, IN2 := 1, ENO => _TMP_EQ23_ENO);
  open_req := _TMP_EQ23_OUT;
  _TMP_EQ24_OUT := EQ(EN := TRUE, IN1 := request, IN2 := 0, ENO => _TMP_EQ24_ENO);
  close_req := _TMP_EQ24_OUT;
END_PROGRAM

CONFIGURATION Config0

  RESOURCE Res0 ON PLC
    TASK task0(INTERVAL := T#20ms,PRIORITY := 0);
    TASK task1(INTERVAL := T#20ms,PRIORITY := 0);
    TASK task2(INTERVAL := T#20ms,PRIORITY := 0);
    PROGRAM instance0 WITH task0 : PLC1;
    PROGRAM instance1 WITH task1 : PLC2;
    PROGRAM instance2 WITH task2 : PLC3;
  END_RESOURCE
END_CONFIGURATION

(* ---- lb_claude_assisted_4e7e2e7a5268_0006.st ---- *)
(*
This code implements a randomly grown symbolic expression:

!(((IN8 & (((xor(xor((xor(xor(IN35 & IN19, !(IN2)), IN2)) & ((xor(xor(IN30, IN50), IN41)) | (!(IN35))), ((IN30 & IN28) & (xor(xor(IN2, IN28), IN4))) & (xor(xor(IN18 | IN27, IN9 & IN35), IN12 & IN6))), xor(xor((IN10 & IN14) & (xor(xor(IN6, IN1), IN48)), xor(xor(IN9, IN41 | IN49), false | IN34)), IN31))) & (!(((false | IN35) & IN15) & IN20))) & (xor(xor(IN9, xor(xor(!(IN25), (IN23 & (IN11 | IN39)) | ((IN39 | IN5) | (!(IN26)))), !(!(!(IN38))))), (!(IN1 | (!(IN31)))) | ((IN14 & IN30) & IN6))))) & (!(xor(xor((xor(xor(((!(IN39)) & (true | IN46)) & ((xor(xor(IN13, IN48), IN49)) | (!(IN43))), IN15), !(xor(xor(IN8 & IN6, xor(xor(IN35, IN42), IN13)), IN48 & IN45)))) & (IN17 & (IN26 | (xor(xor(IN39 & false, IN49), !(IN38))))), xor(xor(xor(xor(!(!(!(IN32))), xor(xor(!(xor(xor(IN41, IN2), IN48)), (IN35 & IN6) | (IN29 & IN32)), xor(xor(!(IN22), xor(xor(IN40, IN4), IN36)), IN23 & IN44))), ((IN35 | IN43) | (!(IN38))) | (!(IN26 | IN25))), !((!(IN33 | IN33)) & (xor(xor(xor(xor(IN25, IN3), IN39), IN40), IN26 | IN49)))), IN9)), IN26)))) | ((!((xor(xor(xor(xor(xor(xor((IN27 & IN28) | (IN45 & IN6), (IN25 & IN38) | (IN23 & IN23)), IN48 & (IN40 | IN29)), xor(xor((xor(xor(IN25, IN11), IN33)) & IN36, !(IN40)), xor(xor(IN47 | IN47, !(IN48)), IN30))), IN3), !((IN42 | IN22) & ((IN13 | IN19) & (!(IN22))))), xor(xor(!(IN41 | (IN38 | IN29)), xor(xor(!(IN6 & IN31), IN28), !(xor(xor(IN41, IN32), IN12)))), ((!(IN22)) | (!(IN2))) & (!(IN40 | false))))) | (xor(xor(xor(xor(((IN47 & IN7) & (!(IN19))) & IN3, (!(IN5 & true)) | (!(IN21 & IN16))), ((!(IN12)) & (xor(xor(IN36, IN38), IN43))) & (!(!(IN1)))), IN13), IN11)))) & (!(!((xor(xor(((!(IN5)) & IN1) & IN43, (IN35 & IN17) | IN39), IN32)) & (!(xor(xor(!(!(IN39)), IN13), xor(xor(!(IN20), IN2 & IN50), xor(xor(IN14, IN3), IN25))))))))))

*)

FUNCTION_BLOCK F_CollectInput
  VAR_IN_OUT
      Data : ARRAY[1..50] OF BOOL;
  END_VAR
  VAR_INPUT
      TICK  : BOOL := 0;
      IN1   : BOOL := 0;
      IN2   : BOOL := 0;
      IN3   : BOOL := 0;
      IN4   : BOOL := 0;
      IN5   : BOOL := 0;
      RESET : BOOL := FALSE;
  END_VAR
  VAR_OUTPUT
      Finished : BOOL;
  END_VAR
  VAR
      j    : USINT := 1;
      tock : BOOL  := 0;
  END_VAR
  IF NOT RESET AND tock = NOT TICK THEN
      Data[j]   := IN1;
      Data[j+1] := IN2;
      Data[j+2] := IN3;
      Data[j+3] := IN4;
      Data[j+4] := IN5;
      j := j + 5;
      tock := TICK;
  ELSE
      j := 1;
      tock := 0;
  END_IF;
  Finished := (j > 50);
END_FUNCTION_BLOCK

PROGRAM Boiler
  VAR
    Data  : ARRAY[1..50] OF BOOL;
    Ready : BOOL;
    CollectInput : F_CollectInput;
  END_VAR
  VAR
    TICK     AT %IX1.0 : BOOL;
    IN1      AT %IX0.3 : BOOL;
    IN2      AT %IX0.4 : BOOL;
    IN3      AT %IX0.5 : BOOL;
    IN4      AT %IX0.6 : BOOL;
    IN5      AT %IX0.7 : BOOL;
    OutReady AT %QX0.0 : BOOL := FALSE;
    FeedNext AT %QX0.1 : BOOL := FALSE;
    Out      AT %QX0.2 : BOOL;
  END_VAR
  CollectInput(TICK:=TICK, IN1:=IN1, IN2:=IN2, IN3:=IN3, IN4:=IN4, IN5:=IN5);
  Ready := CollectInput.Finished;
  FeedNext := 1;
  IF Ready THEN
    Out := (NOT (((Data[8] AND ((((((((Data[35] AND Data[19]) XOR (NOT Data[2])) XOR Data[2]) AND (((Data[30] XOR Data[50]) XOR Data[41]) OR (NOT Data[35]))) XOR (((Data[30] AND Data[28]) AND ((Data[2] XOR Data[28]) XOR Data[4])) AND (((Data[18] OR Data[27]) XOR (Data[9] AND Data[35])) XOR (Data[12] AND Data[6])))) XOR ((((Data[10] AND Data[14]) AND ((Data[6] XOR Data[1]) XOR Data[48])) XOR ((Data[9] XOR (Data[41] OR Data[49])) XOR (FALSE OR Data[34]))) XOR Data[31])) AND (NOT (((FALSE OR Data[35]) AND Data[15]) AND Data[20]))) AND ((Data[9] XOR (((NOT Data[25]) XOR ((Data[23] AND (Data[11] OR Data[39])) OR ((Data[39] OR Data[5]) OR (NOT Data[26])))) XOR (NOT (NOT (NOT Data[38]))))) XOR ((NOT (Data[1] OR (NOT Data[31]))) OR ((Data[14] AND Data[30]) AND Data[6]))))) AND (NOT ((((((((NOT Data[39]) AND (TRUE OR Data[46])) AND (((Data[13] XOR Data[48]) XOR Data[49]) OR (NOT Data[43]))) XOR Data[15]) XOR (NOT (((Data[8] AND Data[6]) XOR ((Data[35] XOR Data[42]) XOR Data[13])) XOR (Data[48] AND Data[45])))) AND (Data[17] AND (Data[26] OR (((Data[39] AND FALSE) XOR Data[49]) XOR (NOT Data[38]))))) XOR (((((NOT (NOT (NOT Data[32]))) XOR (((NOT ((Data[41] XOR Data[2]) XOR Data[48])) XOR ((Data[35] AND Data[6]) OR (Data[29] AND Data[32]))) XOR (((NOT Data[22]) XOR ((Data[40] XOR Data[4]) XOR Data[36])) XOR (Data[23] AND Data[44])))) XOR (((Data[35] OR Data[43]) OR (NOT Data[38])) OR (NOT (Data[26] OR Data[25])))) XOR (NOT ((NOT (Data[33] OR Data[33])) AND ((((Data[25] XOR Data[3]) XOR Data[39]) XOR Data[40]) XOR (Data[26] OR Data[49]))))) XOR Data[9])) XOR Data[26]))) OR ((NOT (((((((((Data[27] AND Data[28]) OR (Data[45] AND Data[6])) XOR ((Data[25] AND Data[38]) OR (Data[23] AND Data[23]))) XOR (Data[48] AND (Data[40] OR Data[29]))) XOR (((((Data[25] XOR Data[11]) XOR Data[33]) AND Data[36]) XOR (NOT Data[40])) XOR (((Data[47] OR Data[47]) XOR (NOT Data[48])) XOR Data[30]))) XOR Data[3]) XOR (NOT ((Data[42] OR Data[22]) AND ((Data[13] OR Data[19]) AND (NOT Data[22]))))) XOR (((NOT (Data[41] OR (Data[38] OR Data[29]))) XOR (((NOT (Data[6] AND Data[31])) XOR Data[28]) XOR (NOT ((Data[41] XOR Data[32]) XOR Data[12])))) XOR (((NOT Data[22]) OR (NOT Data[2])) AND (NOT (Data[40] OR FALSE))))) OR (((((((Data[47] AND Data[7]) AND (NOT Data[19])) AND Data[3]) XOR ((NOT (Data[5] AND TRUE)) OR (NOT (Data[21] AND Data[16])))) XOR (((NOT Data[12]) AND ((Data[36] XOR Data[38]) XOR Data[43])) AND (NOT (NOT Data[1])))) XOR Data[13]) XOR Data[11]))) AND (NOT (NOT ((((((NOT Data[5]) AND Data[1]) AND Data[43]) XOR ((Data[35] AND Data[17]) OR Data[39])) XOR Data[32]) AND (NOT (((NOT (NOT Data[39])) XOR Data[13]) XOR (((NOT Data[20]) XOR (Data[2] AND Data[50])) XOR ((Data[14] XOR Data[3]) XOR Data[25]))))))))));
    OutReady := 1;
    CollectInput(RESET:=TRUE);
  END_IF;
END_PROGRAM

CONFIGURATION Config0
  RESOURCE Res0 ON PLC
    TASK task0(INTERVAL := T#20ms,PRIORITY := 0);
    PROGRAM instance0 WITH task0 : Boiler;
  END_RESOURCE
END_CONFIGURATION

(* ---- lb_claude_assisted_4ea4c0b2d535_0002.st ---- *)
FUNCTION_BLOCK T_PLC_MS_block
	VAR_OUTPUT
		T_PLC_MS :	UDINT;
	END_VAR

	VAR
		PLC_TICKS_PER_SEC :	INT;
		PLC_SYS_TICK_CNT :	DINT;
	END_VAR

	VAR
		debug :	BOOL;(*Debug-Mode ON / OFF*)
		N :	INT;(*Debug-Faktor*)
		Offset :	UDINT;(*Debug-Offset*)
		temp :	DWORD := DWORD#1;(*Debug-Offset*)
		MODE :	BOOL;(*modus*)
		faktor :	UDINT;(*Systemtakt-Faktor*)
		init :	BOOL;
		v_plc_ticks_per_sec :	UDINT;
		base :	UDINT := UDINT#1000;
	END_VAR

	IF init = FALSE THEN
		v_plc_ticks_per_sec := INT_TO_UDINT(PLC_TICKS_PER_SEC);
		IF v_plc_ticks_per_sec = UDINT#1024 THEN
			faktor := UDINT#1;
			MODE := FALSE;
		ELSIF v_plc_ticks_per_sec > UDINT#0 THEN
			IF v_plc_ticks_per_sec <= base THEN
				faktor := base / v_plc_ticks_per_sec;
				MODE := FALSE;
			ELSE
				faktor := v_plc_ticks_per_sec / base;
				MODE := TRUE;
			END_IF;
		ELSE
			faktor := UDINT#1;
		END_IF;
		init := TRUE;
	END_IF;

	IF MODE THEN
		T_PLC_MS := DINT_TO_UDINT(PLC_SYS_TICK_CNT) / faktor;
	ELSE
		T_PLC_MS := DINT_TO_UDINT(PLC_SYS_TICK_CNT) * faktor;
	END_IF;

	IF debug THEN
		T_PLC_MS := (DWORD_TO_UDINT(SHL(UDINT_TO_DWORD(T_PLC_MS),N) OR SHL(temp,N)) - UDINT#1) + Offset;
	END_IF;
END_FUNCTION_BLOCK

FUNCTION_BLOCK INTEGRATE

	VAR_INPUT
		E :	BOOL := TRUE;
		X :	REAL;
		K :	REAL := 1.0;
	END_VAR

	VAR_IN_OUT
		Y :	REAL;
	END_VAR

	VAR
		X_LAST :	REAL;
		init :	BOOL;
		T_PLC_MS :	T_PLC_MS_block;
		last :	UDINT;
		TX :	UDINT;
	END_VAR

	T_PLC_MS();
	TX:= T_PLC_MS.T_PLC_MS;

	IF NOT init THEN
		init := TRUE;
		X_LAST := X;
	ELSIF E THEN
		Y := (X + X_LAST) * 0.5E-3 * UDINT_TO_REAL(TX-last) * K + Y;
		X_LAST := X;
	END_IF;
	last := TX;

END_FUNCTION_BLOCK

FUNCTION_BLOCK FT_INT_Block

	VAR_INPUT
		IN :	REAL;
		K :	REAL := 1.0;
		RUN :	BOOL := TRUE;
		RST :	BOOL;
		OUT_MIN :	REAL := REAL#-1.0E-37;
		OUT_MAX :	REAL := REAL#1.0E37;
	END_VAR

	VAR_OUTPUT
		OUT :	REAL;
		LIM :	BOOL;
	END_VAR

	VAR
		INTEG :	INTEGRATE;
	END_VAR

	IF RST THEN
		OUT := 0.0;
	ELSE
		INTEG(X := IN, E := RUN, K := K, Y := OUT);
		OUT := INTEG.Y;
	END_IF;

	(* limit the OUTputs *)
	IF OUT >= OUT_MAX THEN
		OUT := OUT_MAX;
		LIM := TRUE;
	ELSIF OUT <= OUT_MIN THEN
		OUT := OUT_MIN;
		LIM := TRUE;
	ELSE
		LIM := FALSE;
	END_IF;

END_FUNCTION_BLOCK

FUNCTION_BLOCK FT_PI

	VAR_INPUT
		IN :	REAL;
		KP :	REAL := 1.0;
		KI :	REAL := 1.0;
		ILIM_L :	REAL := -1.0E38;
		ILIM_H :	REAL := 1.0E38;
		IEN :	BOOL := TRUE;
		RST :	BOOL := FALSE;
	END_VAR

	VAR_OUTPUT
		Y :	REAL;
		LIM :	BOOL;
	END_VAR

	VAR
		INTEG :	FT_INT_Block;
	END_VAR

	INTEG(IN := IN, K := KI, RUN := IEN, RST := RST, OUT_MIN := ILIM_L, OUT_MAX := ILIM_H);
	(* check if INTEGrator has reached its limits and set OVERFLOW *)
	LIM := INTEG.LIM;
	Y := KP * IN + INTEG.OUT;

END_FUNCTION_BLOCK

PROGRAM program0
	VAR
		IN :	REAL;
		KP :	REAL := 1.0;
		KI :	REAL := 1.0;
		ILIM_L :	REAL := -1.0E38;
		ILIM_H :	REAL := 1.0E38;
		IEN :	BOOL := TRUE;
		RST :	BOOL := FALSE;

		Y :	REAL;
		LIM :	BOOL;

		func_block : FT_PI;
	END_VAR
	func_block.IN :=IN;
	func_block.KP :=KP;
	func_block.KI :=KI;
	func_block.ILIM_L :=ILIM_L;
	func_block.ILIM_H :=ILIM_H;
	func_block.IEN :=IEN;
	func_block.RST :=RST;

	func_block();
	Y := func_block.Y;
	LIM := func_block.LIM;
END_PROGRAM

(* ---- lb_claude_assisted_4f5143802709_0002.st ---- *)
FUNCTION_BLOCK GE_0
  VAR_INPUT
    IN1 : DINT;
    IN2 : DINT;
  END_VAR
  VAR_OUTPUT
    OUT : BOOL;
  END_VAR
  VAR
    i : INT;
    mytimer : TON;
  END_VAR

  OUT:=FALSE;
  IF IN1>=IN2 then
    OUT:=TRUE;
  END_IF;

  mytimer(IN := TRUE, PT := t#8000ms);
  i:=0;
  IF mytimer.Q = TRUE then
     WHILE i<4 do
      OUT:=TRUE;
    End_WHILE;
  End_IF;
END_FUNCTION_BLOCK

PROGRAM PLC3
  VAR_INPUT
    level : DINT;
  END_VAR
  VAR_OUTPUT
    pump : BOOL;
  END_VAR
  VAR
    low : BOOL;
    high : BOOL;
    low_3 : DINT := 0;
    high_3 : DINT := 10;
    GE_00 : GE_0;
    _TMP_LE13_ENO : BOOL;
    _TMP_LE13_OUT : BOOL;
  END_VAR

  GE_00(EN := TRUE, IN1 := level, IN2 := high_3);
  high := GE_00.OUT;
  _TMP_LE13_OUT := LE(EN := TRUE, IN1 := level, IN2 := low_3, ENO => _TMP_LE13_ENO);
  low := _TMP_LE13_OUT;
  pump := NOT(low) AND (high OR pump);
END_PROGRAM

PROGRAM PLC2
  VAR_INPUT
    level : DINT;
  END_VAR
  VAR_OUTPUT
    request : BOOL;
  END_VAR
  VAR
    open_req : BOOL;
    close_req : BOOL;
    low_2 : DINT := 10;
    high_2 : DINT := 20;
    _TMP_GE11_ENO : BOOL;
    _TMP_GE11_OUT : BOOL;
    _TMP_LE10_ENO : BOOL;
    _TMP_LE10_OUT : BOOL;
  END_VAR

  _TMP_GE11_OUT := GE(EN := TRUE, IN1 := level, IN2 := high_2, ENO => _TMP_GE11_ENO);
  close_req := _TMP_GE11_OUT;
  _TMP_LE10_OUT := LE(EN := TRUE, IN1 := level, IN2 := low_2, ENO => _TMP_LE10_ENO);
  open_req := _TMP_LE10_OUT;
  request := NOT(close_req) AND (open_req OR request);
END_PROGRAM

PROGRAM PLC1
  VAR_INPUT
    level : DINT;
    request : DINT;
  END_VAR
  VAR_OUTPUT
    pumps : BOOL;
    valve : BOOL;
  END_VAR
  VAR
    low : BOOL;
    high : BOOL;
    open_req : BOOL;
    close_req : BOOL;
    low_1 : DINT := 40;
    high_1 : DINT := 80;
    _TMP_LE3_ENO : BOOL;
    _TMP_LE3_OUT : BOOL;
    _TMP_GE31_ENO : BOOL;
    _TMP_GE31_OUT : BOOL;
    _TMP_EQ23_ENO : BOOL;
    _TMP_EQ23_OUT : BOOL;
    _TMP_EQ24_ENO : BOOL;
    _TMP_EQ24_OUT : BOOL;
  END_VAR

  _TMP_LE3_OUT := LE(EN := TRUE, IN1 := level, IN2 := low_1, ENO => _TMP_LE3_ENO);
  low := _TMP_LE3_OUT;
  _TMP_GE31_OUT := GE(EN := TRUE, IN1 := level, IN2 := high_1, ENO => _TMP_GE31_ENO);
  high := _TMP_GE31_OUT;
  pumps := NOT(high) AND (low OR pumps);
  valve := NOT(close_req) AND (valve OR open_req AND NOT(low));
  _TMP_EQ23_OUT := EQ(EN := TRUE, IN1 := request, IN2 := 1, ENO => _TMP_EQ23_ENO);
  open_req := _TMP_EQ23_OUT;
  _TMP_EQ24_OUT := EQ(EN := TRUE, IN1 := request, IN2 := 0, ENO => _TMP_EQ24_ENO);
  close_req := _TMP_EQ24_OUT;
END_PROGRAM

CONFIGURATION Config0

  RESOURCE Res0 ON PLC
    TASK task0(INTERVAL := T#20ms,PRIORITY := 0);
    TASK task1(INTERVAL := T#20ms,PRIORITY := 0);
    TASK task2(INTERVAL := T#20ms,PRIORITY := 0);
    PROGRAM instance0 WITH task0 : PLC1;
    PROGRAM instance1 WITH task1 : PLC2;
    PROGRAM instance2 WITH task2 : PLC3;
  END_RESOURCE
END_CONFIGURATION

(* ---- lb_claude_assisted_5359f367f65f_0011.st ---- *)
FUNCTION_BLOCK TOOL_CHANGER

VAR_INPUT
    ToolChangeRequired : BOOL; (** True if tool change is required **)
    ToolCarouselPosition : INT; (** Current position of the tool carousel **)
    DesiredToolNumber : INT; (** Number of the desired tool **)
END_VAR

VAR_OUTPUT
    RotateCarousel : BOOL; (** Rotate the tool carousel **)
    LockTool : BOOL; (** Lock the tool in the spindle **)
END_VAR

VAR
    ToolChangeState : INT; (**0=Idle, 1=RotatingCarousel, 2=LockingTool**)
END_VAR

IF ToolChangeRequired THEN
    CASE ToolChangeState OF
        0:
            (** Check if carousel needs to rotate **)
            IF ToolCarouselPosition <> DesiredToolNumber THEN
                RotateCarousel := TRUE;
                ToolChangeState := 1;
            ELSE
                LockTool := TRUE;
                ToolChangeState := 2;
            END_IF;

        1:
            (** Wait for carousel to reach desired position **)
            IF ToolCarouselPosition = DesiredToolNumber THEN
                RotateCarousel := FALSE;
                LockTool := TRUE;
                ToolChangeState := 2;
            END_IF;

        2:
            (** Wait for tool to be locked **)
            LockTool := FALSE;
            ToolChangeState := 0;
    END_CASE;
END_IF;

END_FUNCTION_BLOCK

(* ---- lb_claude_assisted_55fbc4d881a4_0037.st ---- *)
FUNCTION_BLOCK StackMin
VAR_INPUT
    push : BOOL;
    pop : BOOL;
    reset : BOOL;
END_VAR
VAR_OUTPUT
    error : BOOL;
    status : WORD;
END_VAR
VAR_IN_OUT
    item : INT;
    stack : ARRAY[0..3] OF INT;
END_VAR
VAR
    top : INT := -1;
    min_index : INT;
    i : INT;
    temp_min : INT;
END_VAR

(* Reset has highest priority *)
IF reset THEN
    top := -1;
    error := FALSE;
    status := 16#0000;
(* Push operation *)
ELSIF push THEN
    IF top = 3 THEN
        error := TRUE;
        status := 16#8A04;
    ELSE
        top := top + 1;
        stack[top] := item;
        error := FALSE;
        status := 16#0000;
    END_IF;
(* Pop operation *)
ELSIF pop THEN
    IF top = -1 THEN
        error := TRUE;
        status := 16#8A05;
    ELSE
        (* Find minimum value and its index *)
        min_index := 0;
        temp_min := stack[0];
        FOR i := 1 TO top DO
            IF stack[i] < temp_min THEN
                temp_min := stack[i];
                min_index := i;
            END_IF;
        END_FOR;

        (* Store min value in output *)
        item := temp_min;

        (* Shift elements down *)
        FOR i := min_index TO top - 1 DO
            stack[i] := stack[i + 1];
        END_FOR;

        (* Decrement top *)
        top := top - 1;
        error := FALSE;
        status := 16#0000;
    END_IF;
(* No operation - clear error state *)
ELSE
    error := FALSE;
    status := 16#0000;
END_IF;
END_FUNCTION_BLOCK

(* ---- lb_claude_assisted_56c02a912be6_0076.st ---- *)
FUNCTION UDINT_TO_TIME2:TIME

	VAR_INPUT
		IN :	UDINT;
	END_VAR

	UDINT_TO_TIME2 := DINT_TO_TIME(UDINT_TO_DINT(IN));

END_FUNCTION

FUNCTION_BLOCK T_PLC_MS_block
	VAR_OUTPUT
		T_PLC_MS :	UDINT;
	END_VAR

	VAR_EXTERNAL
		PLC_TICKS_PER_SEC :	INT;
		PLC_SYS_TICK_CNT :	DINT;
	END_VAR

	VAR
		debug :	BOOL;(*Debug-Mode ON / OFF*)
		N :	INT;(*Debug-Faktor*)
		Offset :	UDINT;(*Debug-Offset*)
		temp :	DWORD := DWORD#1;(*Debug-Offset*)
		mode :	BOOL;(*modus*)
		faktor :	UDINT;(*Systemtakt-Faktor*)
		init :	BOOL;
		v_plc_ticks_per_sec :	UDINT;
		base :	UDINT := UDINT#1000;
	END_VAR

	IF init = FALSE THEN
		v_plc_ticks_per_sec := INT_TO_UDINT(PLC_TICKS_PER_SEC);
		IF v_plc_ticks_per_sec = UDINT#1024 THEN
			faktor := UDINT#1;
			mode := FALSE;
		ELSIF v_plc_ticks_per_sec > UDINT#0 THEN
			IF v_plc_ticks_per_sec <= base THEN
				faktor := base / v_plc_ticks_per_sec;
				mode := FALSE;
			ELSE
				faktor := v_plc_ticks_per_sec / base;
				mode := TRUE;
			END_IF;
		ELSE
			faktor := UDINT#1;
		END_IF;
		init := TRUE;
	END_IF;

	IF mode THEN
		T_PLC_MS := DINT_TO_UDINT(PLC_SYS_TICK_CNT) / faktor;
	ELSE
		T_PLC_MS := DINT_TO_UDINT(PLC_SYS_TICK_CNT) * faktor;
	END_IF;

	IF debug THEN
		T_PLC_MS := (DWORD_TO_UDINT(SHL(UDINT_TO_DWORD(T_PLC_MS),N) OR SHL(temp,N)) - UDINT#1) + Offset;
	END_IF;

END_FUNCTION_BLOCK

FUNCTION TIME_TO_UDINT2:UDINT
	VAR_INPUT
		X :	TIME;
	END_VAR

	TIME_TO_UDINT2 := DINT_TO_UDINT(TIME_TO_DINT(X));
END_FUNCTION

FUNCTION FRMP_B:BYTE
	VAR_INPUT
		START :	BYTE;
		DIR :	BOOL;
		TD :	TIME;
		TR :	TIME;
	END_VAR

	IF TD < TR THEN
		FRMP_B := MIN(UDINT_TO_BYTE(DWORD_TO_UDINT(SHL(TIME_TO_DWORD(TD), 8)) / TIME_TO_UDINT2(TR)), SEL(DIR, START, USINT_TO_BYTE(USINT#255 - BYTE_TO_USINT(START))));
		IF DIR THEN
			FRMP_B := USINT_TO_BYTE(BYTE_TO_USINT(START) + BYTE_TO_USINT(FRMP_B));
		ELSE
			FRMP_B := USINT_TO_BYTE(BYTE_TO_USINT(START) - BYTE_TO_USINT(FRMP_B));
		END_IF;
	ELSE
		FRMP_B := SEL(DIR, BYTE#0, BYTE#255);
	END_IF;
END_FUNCTION

FUNCTION_BLOCK _RMP_B
	VAR_INPUT
		DIR :	BOOL;
		E :	BOOL := TRUE;
		TR :	TIME;
	END_VAR

	VAR_IN_OUT
		RMP :	BYTE;
	END_VAR

	VAR
		T_PLC_MS :	T_PLC_MS_Block;
		tx :	TIME;
		tl :	TIME;
		tn :	TIME;
		init :	BOOL;
		last_dir :	BOOL;
		start :	BYTE;
	END_VAR

	T_PLC_MS();
	tx := UDINT_TO_TIME(T_PLC_MS.T_PLC_MS);

	IF E AND init AND (dir = last_dir) AND (RMP <> SEL(DIR, BYTE#0, BYTE#255)) AND TR = tn THEN
		RMP := FRMP_B(start, DIR, tx - tl, TR);
	ELSE
		init := TRUE;
		tl := tx;
		tn := tr;
		start := RMP;
	END_IF;
	last_dir := dir;
END_FUNCTION_BLOCK

FUNCTION_BLOCK CLICK_MODE_Block

	VAR_INPUT
		IN :	BOOL;
		T_LONG :	TIME := T#500ms;
	END_VAR

	VAR_OUTPUT
		SINGLE :	BOOL;
		DOUBLE :	BOOL;
		LONG :	BOOL;
		TP_LONG :	BOOL;
	END_VAR

	VAR
		Timer :	TP;
		cnt :	INT;
		last :	BOOL;
	END_VAR

	timer(in := IN, PT := T_LONG);
	single := FALSE;
	double := FALSE;

	IF timer.Q THEN
		IF NOT in AND last THEN	cnt := cnt + 1; END_IF;
	ELSE
		CASE cnt OF
			1 : single := TRUE;
			2 : double := TRUE;
		END_CASE;
		cnt := 0;
	END_IF;
	last := in;
	TP_LONG := NOT timer.Q AND (NOT LONG) AND IN;
	LONG := NOT timer.Q AND in;

END_FUNCTION_BLOCK

FUNCTION_BLOCK DIMM_2_Block

	VAR_INPUT
		SET :	BOOL;
		VAL :	BYTE := BYTE#255;
		I1 :	BOOL;
		I2 :	BOOL;
		RST :	BOOL;
		T_DEBOUNCE :	TIME := T#10ms;
		T_ON_MAX :	TIME := T#0h;
		T_DIMM_START :	TIME := T#1s;
		T_DIMM :	TIME := T#3s;
		MIN_ON :	BYTE := BYTE#50;
		MAX_ON :	BYTE := BYTE#255;
		RST_OUT :	BOOL;
		SOFT_DIMM :	BOOL := TRUE;
		DBL1_TOG :	BOOL;
		DBL2_TOG :	BOOL;
		DBL1_SET :	BOOL;
		DBL2_SET :	BOOL;
		DBL1_POS :	BYTE;
		DBL2_POS :	BYTE;
	END_VAR

	VAR_OUTPUT
		Q :	BOOL;
		D1 :	BOOL;
		D2 :	BOOL;
	END_VAR

	VAR_IN_OUT
		_OUT :	BYTE;
	END_VAR

	VAR
		t1 :	TOF;
		t2 :	TOF;
		dc1 :	CLICK_MODE_Block;
		dc2 :	CLICK_MODE_Block;
		t3 :	TON;
		dim :	_RMP_B;
	END_VAR

	t1(IN := I1, PT := T_DEBOUNCE);
	t2(IN := I2, PT := T_DEBOUNCE);
	dc1(in := t1.Q, T_LONG := T_DIMM_START);
	dc2(in := t2.Q, T_LONG := T_DIMM_START);

	IF RST THEN
		IF RST_OUT THEN _OUT := BYTE#0; END_IF;
		Q := FALSE;
		D1 := FALSE;
		D2 := FALSE;
	ELSIF set THEN
		_OUT := VAL;
		Q := TRUE;
	ELSIF dc1.SINGLE THEN
		_OUT := LIMIT(MAX(MIN_ON,BYTE#1), _OUT, MAX_ON);
		Q := TRUE;
	ELSIF dc2.SINGLE THEN
		Q := FALSE;
	ELSIF dc1.TP_LONG THEN
		IF NOT Q THEN
			_OUT := SEL(SOFT_DIMM, LIMIT(MAX(MIN_ON,BYTE#1), _OUT, MAX_ON), BYTE#1);
		END_IF;
		Q := TRUE;
		dim.DIR := TRUE;
	ELSIF dc2.TP_LONG THEN
		dim.DIR := FALSE;
	END_IF;

	IF NOT DBL1_TOG THEN D1 := FALSE; END_IF;
	IF dc1.DOUBLE THEN
		IF DBL1_SET THEN
			_OUT := DBL1_POS;
			Q := TRUE;
		ELSE
			D1 := NOT D1;
		END_IF;
	END_IF;
	IF NOT DBL2_TOG THEN D2 := FALSE; END_IF;
	IF dc2.DOUBLE THEN
		IF DBL2_SET THEN
			_OUT := DBL2_POS;
			Q := TRUE;
		ELSE
			D2 := NOT D2;
		END_IF;
	END_IF;

	dim(dir := dc2.LONG, e := dc1.LONG OR dc2.LONG , TR := T_DIMM, rmp := _OUT);
	_OUT := dim.RMP;

	IF _OUT = BYTE#0 THEN Q := FALSE; END_IF;

	IF t_ON_MAX > t#0s THEN
		t3(in := q, pt := T_ON_MAX);
		Q := Q XOR t3.Q;
	END_IF;

END_FUNCTION_BLOCK

PROGRAM program0
	VAR
	    SET :	BOOL;
		VAL :	BYTE := BYTE#255;
		I1 :	BOOL;
		I2 :	BOOL;
		RST :	BOOL;
		T_DEBOUNCE :	TIME := T#10ms;
		T_ON_MAX :	TIME := T#0h;
		T_DIMM_START :	TIME := T#1s;
		T_DIMM :	TIME := T#3s;
		MIN_ON :	BYTE := BYTE#50;
		MAX_ON :	BYTE := BYTE#255;
		RST_OUT :	BOOL;
		SOFT_DIMM :	BOOL := TRUE;
		DBL1_TOG :	BOOL;
		DBL2_TOG :	BOOL;
		DBL1_SET :	BOOL;
		DBL2_SET :	BOOL;
		DBL1_POS :	BYTE;
		DBL2_POS :	BYTE;
		_OUT :	BYTE := BYTE#0;
		Q :	BOOL;
		D1 :	BOOL;
		D2 :	BOOL;

		func_block : DIMM_2_Block;
  	END_VAR
	func_block.SET := SET;
	func_block.VAL := VAL;
	func_block.I1 := I1;
	func_block.I2 := I2;
	func_block.RST := RST;
	func_block.T_DEBOUNCE := T_DEBOUNCE;
	func_block.T_ON_MAX := T_ON_MAX;
	func_block.T_DIMM_START := T_DIMM_START;
	func_block.T_DIMM := T_DIMM;
	func_block.MIN_ON := MIN_ON;
	func_block.MAX_ON := MAX_ON;
	func_block.RST_OUT := RST_OUT;
	func_block.SOFT_DIMM := SOFT_DIMM;
	func_block.DBL1_TOG := DBL1_TOG;
	func_block.DBL2_TOG := DBL2_TOG;
	func_block.DBL1_SET := DBL1_SET;
	func_block.DBL2_SET := DBL2_SET;
	func_block.DBL1_POS := DBL1_POS;
	func_block.DBL2_POS := DBL2_POS;
	func_block._OUT := _OUT;

	func_block();
	_OUT := func_block._OUT;
	Q := func_block.Q;
	D1 := func_block.D1;
	D2 := func_block.D2;
END_PROGRAM

CONFIGURATION Config0
	VAR_GLOBAL
		PLC_TICKS_PER_SEC :	INT;
		PLC_SYS_TICK_CNT :	DINT;
	END_VAR
  	RESOURCE Res0 ON PLC
    	TASK task0(INTERVAL := T#20ms,PRIORITY := 0);
    	PROGRAM instance0 WITH task0 : program0;
  	END_RESOURCE
END_CONFIGURATION

(* ---- lb_claude_assisted_57c656b059c7_0013.st ---- *)
(*
This code implements a randomly grown symbolic expression:

(IN21 & (xor(xor(((IN15 | (xor(xor(((xor(xor(IN46, IN46), IN48)) & (IN48 & IN37)) | (xor(xor(IN13 & IN17, IN18 | IN36), IN43)), (!(IN20 & IN16)) & (true & IN10)), xor(xor((IN8 & IN24) & (IN6 | IN40), (IN20 | IN43) & (!(IN22))), IN27 & (IN16 & IN29))))) | (IN7 & IN37)) | ((xor(xor(IN49, IN22), ((!(!(IN10))) & IN12) & (((IN2 | IN15) | (IN30 | IN34)) | (!(IN42 & IN45))))) & ((!(xor(xor(IN33 & IN39, (IN12 & IN13) & (IN8 | IN38)), (!(IN4)) | (!(IN49))))) | (!(!((IN44 | IN30) & IN11))))), xor(xor(((!(xor(xor(IN49 | (IN16 | IN40), (IN21 | IN13) & IN42), !(IN49 & IN21)))) | IN48) | (xor(xor(IN9, (((IN32 | IN17) & (!(IN31))) & ((!(IN28)) & (IN43 | IN29))) & (true & ((xor(xor(false, IN29), IN12)) & (IN14 & IN39)))), !(!(xor(xor(IN17, !(IN48)), IN15 & IN25))))), IN29), (((xor(xor(xor(xor(IN40, IN33 & IN22), IN31 | IN14), IN27), (!(IN9)) & (xor(xor(IN25, IN49), IN10)))) | ((xor(xor(!(IN2), IN1), IN6 & IN12)) | IN35)) | ((xor(xor(IN27, !(!(IN28))), IN33)) & (!((!(IN11)) | (!(IN46)))))) | (xor(xor(IN28, IN39), !(xor(xor(!(IN49), xor(xor(xor(xor(IN46, IN9), IN37), IN36), IN35 | IN27)), xor(xor(IN8 | IN24, IN20 & IN28), IN20))))))), IN25))) & IN46

*)

FUNCTION_BLOCK F_CollectInput
  VAR_IN_OUT
      Data : ARRAY[1..50] OF BOOL;
  END_VAR
  VAR_INPUT
      TICK  : BOOL := 0;
      IN1   : BOOL := 0;
      IN2   : BOOL := 0;
      IN3   : BOOL := 0;
      IN4   : BOOL := 0;
      IN5   : BOOL := 0;
      RESET : BOOL := FALSE;
  END_VAR
  VAR_OUTPUT
      Finished : BOOL;
  END_VAR
  VAR
      j    : USINT := 1;
      tock : BOOL  := 0;
  END_VAR
  IF NOT RESET AND tock = NOT TICK THEN
      Data[j]   := IN1;
      Data[j+1] := IN2;
      Data[j+2] := IN3;
      Data[j+3] := IN4;
      Data[j+4] := IN5;
      j := j + 5;
      tock := TICK;
  ELSE
      j := 1;
      tock := 0;
  END_IF;
  Finished := (j > 50);
END_FUNCTION_BLOCK

PROGRAM Boiler
  VAR
    Data  : ARRAY[1..50] OF BOOL;
    Ready : BOOL;
    CollectInput : F_CollectInput;
  END_VAR
  VAR
    TICK     AT %IX1.0 : BOOL;
    IN1      AT %IX0.3 : BOOL;
    IN2      AT %IX0.4 : BOOL;
    IN3      AT %IX0.5 : BOOL;
    IN4      AT %IX0.6 : BOOL;
    IN5      AT %IX0.7 : BOOL;
    OutReady AT %QX0.0 : BOOL := FALSE;
    FeedNext AT %QX0.1 : BOOL := FALSE;
    Out      AT %QX0.2 : BOOL;
  END_VAR
  CollectInput(TICK:=TICK, IN1:=IN1, IN2:=IN2, IN3:=IN3, IN4:=IN4, IN5:=IN5);
  Ready := CollectInput.Finished;
  FeedNext := 1;
  IF Ready THEN
    Out := ((Data[21] AND (((((Data[15] OR ((((((Data[46] XOR Data[46]) XOR Data[48]) AND (Data[48] AND Data[37])) OR (((Data[13] AND Data[17]) XOR (Data[18] OR Data[36])) XOR Data[43])) XOR ((NOT (Data[20] AND Data[16])) AND (TRUE AND Data[10]))) XOR ((((Data[8] AND Data[24]) AND (Data[6] OR Data[40])) XOR ((Data[20] OR Data[43]) AND (NOT Data[22]))) XOR (Data[27] AND (Data[16] AND Data[29]))))) OR (Data[7] AND Data[37])) OR (((Data[49] XOR Data[22]) XOR (((NOT (NOT Data[10])) AND Data[12]) AND (((Data[2] OR Data[15]) OR (Data[30] OR Data[34])) OR (NOT (Data[42] AND Data[45]))))) AND ((NOT (((Data[33] AND Data[39]) XOR ((Data[12] AND Data[13]) AND (Data[8] OR Data[38]))) XOR ((NOT Data[4]) OR (NOT Data[49])))) OR (NOT (NOT ((Data[44] OR Data[30]) AND Data[11])))))) XOR (((((NOT (((Data[49] OR (Data[16] OR Data[40])) XOR ((Data[21] OR Data[13]) AND Data[42])) XOR (NOT (Data[49] AND Data[21])))) OR Data[48]) OR ((Data[9] XOR ((((Data[32] OR Data[17]) AND (NOT Data[31])) AND ((NOT Data[28]) AND (Data[43] OR Data[29]))) AND (TRUE AND (((FALSE XOR Data[29]) XOR Data[12]) AND (Data[14] AND Data[39]))))) XOR (NOT (NOT ((Data[17] XOR (NOT Data[48])) XOR (Data[15] AND Data[25])))))) XOR Data[29]) XOR (((((((Data[40] XOR (Data[33] AND Data[22])) XOR (Data[31] OR Data[14])) XOR Data[27]) XOR ((NOT Data[9]) AND ((Data[25] XOR Data[49]) XOR Data[10]))) OR ((((NOT Data[2]) XOR Data[1]) XOR (Data[6] AND Data[12])) OR Data[35])) OR (((Data[27] XOR (NOT (NOT Data[28]))) XOR Data[33]) AND (NOT ((NOT Data[11]) OR (NOT Data[46]))))) OR ((Data[28] XOR Data[39]) XOR (NOT (((NOT Data[49]) XOR ((((Data[46] XOR Data[9]) XOR Data[37]) XOR Data[36]) XOR (Data[35] OR Data[27]))) XOR (((Data[8] OR Data[24]) XOR (Data[20] AND Data[28])) XOR Data[20]))))))) XOR Data[25])) AND Data[46]);
    OutReady := 1;
    CollectInput(RESET:=TRUE);
  END_IF;
END_PROGRAM

CONFIGURATION Config0
  RESOURCE Res0 ON PLC
    TASK task0(INTERVAL := T#20ms,PRIORITY := 0);
    PROGRAM instance0 WITH task0 : Boiler;
  END_RESOURCE
END_CONFIGURATION

(* ---- lb_claude_assisted_581056208788_0012.st ---- *)
FUNCTION_BLOCK ONTIME_Block

	VAR_INPUT
		IN :	BOOL;
		RST :	BOOL;
	END_VAR

	VAR_IN_OUT
		SECONDS :	UDINT;
		CYCLES :	UDINT;
	END_VAR

	VAR
		tx :	UDINT;
		last :	UDINT;
		edge :	BOOL;
		init :	BOOL;
		ms :	UDINT;
		T_PLC_MS :	T_PLC_MS_Block;
	END_VAR

	T_PLC_MS();
	tx:= T_PLC_MS.T_PLC_MS;

	IF NOT init THEN
		init := TRUE;
		last := tx;
		ms := UDINT#0;
	END_IF;
	IF RST THEN
		SECONDS := UDINT#0;
		CYCLES := UDINT#0;
		last := tx;
		ms := UDINT#0;
	ELSIF IN THEN
		(* add the current milliseconds *)
		ms := (tx - last) + ms;
		IF ms >= UDINT#1000 THEN
			seconds := seconds + UDINT#1;
			ms := ms - UDINT#1000;
		END_IF;
		cycles := cycles + BOOL_TO_UDINT(NOT edge);
	END_IF;
	last := tx;
	edge := in;

END_FUNCTION_BLOCK

FUNCTION UDINT_TO_TIME2:TIME

	VAR_INPUT
		IN :	UDINT;
	END_VAR

	UDINT_TO_TIME2 := DINT_TO_TIME(UDINT_TO_DINT(IN));

END_FUNCTION

FUNCTION_BLOCK T_PLC_MS_block
	VAR_OUTPUT
		T_PLC_MS :	UDINT;
	END_VAR

	VAR_EXTERNAL
		PLC_TICKS_PER_SEC :	INT;
		PLC_SYS_TICK_CNT :	DINT;
	END_VAR

	VAR
		debug :	BOOL;(*Debug-Mode ON / OFF*)
		N :	INT;(*Debug-Faktor*)
		Offset :	UDINT;(*Debug-Offset*)
		temp :	DWORD := DWORD#1;(*Debug-Offset*)
		mode :	BOOL;(*modus*)
		faktor :	UDINT;(*Systemtakt-Faktor*)
		init :	BOOL;
		v_plc_ticks_per_sec :	UDINT;
		base :	UDINT := UDINT#1000;
	END_VAR

	IF init = FALSE THEN
		v_plc_ticks_per_sec := INT_TO_UDINT(PLC_TICKS_PER_SEC);
		IF v_plc_ticks_per_sec = UDINT#1024 THEN
			faktor := UDINT#1;
			mode := FALSE;
		ELSIF v_plc_ticks_per_sec > UDINT#0 THEN
			IF v_plc_ticks_per_sec <= base THEN
				faktor := base / v_plc_ticks_per_sec;
				mode := FALSE;
			ELSE
				faktor := v_plc_ticks_per_sec / base;
				mode := TRUE;
			END_IF;
		ELSE
			faktor := UDINT#1;
		END_IF;
		init := TRUE;
	END_IF;

	IF mode THEN
		T_PLC_MS := DINT_TO_UDINT(PLC_SYS_TICK_CNT) / faktor;
	ELSE
		T_PLC_MS := DINT_TO_UDINT(PLC_SYS_TICK_CNT) * faktor;
	END_IF;

	IF debug THEN
		T_PLC_MS := (DWORD_TO_UDINT(SHL(UDINT_TO_DWORD(T_PLC_MS),N) OR SHL(temp,N)) - UDINT#1) + Offset;
	END_IF;

END_FUNCTION_BLOCK

FUNCTION_BLOCK BURNER_Block

	VAR_INPUT
		IN :	BOOL;
		STAGE2 :	BOOL;
		OVER_TEMP :	BOOL;
		OIL_TEMP :	BOOL := TRUE;
		FLAME :	BOOL;
		RST :	BOOL;
		RST_TIMER :	BOOL;
		PRE_HEAT_TIME :	TIME := t#5s;
		PRE_VENT_TIME :	TIME := t#15s;
		PRE_IGNITE_TIME :	TIME := t#5s;
		POST_IGNITE_TIME :	TIME := t#25s;
		STAGE2_DELAY :	TIME := t#10s;
		SAFETY_TIME :	TIME := t#5s;
		LOCKOUT_TIME :	TIME := t#10s;
		MULTIPLE_IGNITION :	BOOL := TRUE;
		KW1 :	REAL;
		KW2 :	REAL;
	END_VAR

	VAR_OUTPUT
		MOTOR :	BOOL;
		COIL1 :	BOOL;
		COIL2 :	BOOL;
		PRE_HEAT :	BOOL;
		IGNITE :	BOOL;
		KWH :	REAL;
		STATUS :	BYTE;
		FAIL :	BOOL;
	END_VAR

	VAR_IN_OUT
		RUNTIME1 :	UDINT;
		RUNTIME2 :	UDINT;
		CYCLES :	UDINT;
	END_VAR

	VAR
		state :	INT;
		last :	TIME;
		tx :	TIME;
		last_change :	TIME;
		timer1 :	ONTIME_Block;
		timer2 :	ONTIME_Block;
		oil_temp_last :	BOOL;
		cycles2 :	UDINT;
		T_PLC_MS :	T_PLC_MS_Block;
	END_VAR

	T_PLC_MS();
	tx:= UDINT_TO_TIME(T_PLC_MS.T_PLC_MS);

	IF rst OR over_temp OR state = 0 THEN
		IF status > BYTE#0 AND tx - last_change >= lockout_time AND rst THEN
			status := BYTE#110;
			fail := FALSE;
			state := 1;
		ELSE
			motor := FALSE;
			coil1 := FALSE;
			coil2 := FALSE;
			ignite := FALSE;
			pre_heat := FALSE;
			IF over_temp THEN
				status := BYTE#9;
				fail := TRUE;
			END_IF;
			last_change := tx;
			last := tx;
			state := 1;
		END_IF;
	END_IF;

	IF rst_timer THEN
		runtime1 := UDINT#0;
		runtime2 := UDINT#0;
		cycles := UDINT#0;
		cycles2 := UDINT#0;
	END_IF;

	IF (status > BYTE#0 AND status < BYTE#100) OR rst THEN RETURN; END_IF;

	CASE state OF

	1:
		IF in AND flame THEN
			state := 7;
			pre_heat := FALSE;
			status := BYTE#2;
			last_change := tx;
		ELSIF in THEN
			pre_heat := TRUE;
			state := 2;
			last_change := tx;
		END_IF;

	2:
		IF (tx- last_change >= pre_heat_time AND oil_temp) OR (oil_temp AND NOT oil_temp_last) THEN
			motor := TRUE;
			state := 3;
			last_change := tx;
		ELSIF tx - last_change >= pre_heat_time AND NOT oil_temp THEN
			state := 7;
			pre_heat := FALSE;
			status := BYTE#1;
			last_change := tx;
		ELSIF flame THEN
			state := 7;
			pre_heat := FALSE;
			status := BYTE#2;
			last_change := tx;
		END_IF;

	3:
		IF tx - last_change >= pre_vent_time - pre_ignite_time THEN
			ignite := TRUE;
			state := 4;
			last_change := tx;
		ELSIF flame THEN
			state := 7;
			pre_heat := FALSE;
			motor := FALSE;
			status := BYTE#3;
			last_change := tx;
		END_IF;

	4:
		IF tx - last_change >= pre_ignite_time THEN
			coil1 := TRUE;
			state := 5;
			last_change := tx;
		END_IF;

	5:
		IF tx - last_change >= safety_time OR flame THEN
			IF NOT flame THEN
				state := 7;
				motor := FALSE;
				coil1 := FALSE;
				pre_heat := FALSE;
				ignite := FALSE;
				status := BYTE#4;
				last_change := tx;
			ELSE
				state := 6;
				last_change := tx;
			END_IF;
		END_IF;

	6:
		IF NOT flame AND NOT multiple_ignition THEN
			state := 7;
			motor := FALSE;
			coil1 := FALSE;
			coil2 := FALSE;
			pre_heat := FALSE;
			ignite := FALSE;
			status := BYTE#5;
			last_change := tx;
		ELSIF NOT flame AND multiple_ignition THEN
			ignite := TRUE;
			state := 5;
			coil2 := FALSE;
			last_change := tx;
		ELSE
			IF tx - last_change >= post_ignite_time THEN
				ignite := FALSE;
			END_IF;
			IF tx - last_change >= stage2_delay AND stage2 THEN
				coil2 := TRUE;
			ELSE
				coil2 := FALSE;
			END_IF;
		END_IF;
	END_CASE;

	IF NOT in THEN
		state := 1;
		motor := FALSE;
		coil1 := FALSE;
		coil2 := FALSE;
		ignite := FALSE;
		pre_heat := FALSE;
		last_change := tx;
	END_IF;

	timer1(in := flame AND in AND motor AND coil1 AND NOT coil2, SECONDS := runtime1, CYCLES := cycles);
	cycles := timer1.CYCLES;
	runtime1 := timer1.SECONDS;

	timer2(in := flame AND in AND motor AND coil1 AND coil2, SECONDS := runtime2, CYCLES := cycles2);
	cycles2 := timer2.CYCLES;
	runtime2 := timer2.SECONDS;

	KWH := UDINT_TO_REAL(runtime1) * KW1 / 3600.0 + UDINT_TO_REAL(runtime2) * KW2 / 3600.0;

	last := tx;

	IF status > BYTE#0 AND status < BYTE#100 THEN
		fail := TRUE;
	ELSE
		fail := FALSE;
		IF NOT in THEN
			status := BYTE#110;
		ELSIF flame AND in AND motor AND coil2 AND coil1 THEN
			status := BYTE#113;
		ELSIF flame AND in AND motor AND coil1 THEN
			status := BYTE#112;
		ELSE
			status := BYTE#111;
		END_IF;
	END_IF;

END_FUNCTION_BLOCK

PROGRAM program0
	VAR
		IN :	BOOL;
		STAGE2 :	BOOL;
		OVER_TEMP :	BOOL;
		OIL_TEMP :	BOOL := TRUE;
		FLAME :	BOOL;
		RST :	BOOL;
		RST_TIMER :	BOOL;
		PRE_HEAT_TIME :	TIME := t#5s;
		PRE_VENT_TIME :	TIME := t#15s;
		PRE_IGNITE_TIME :	TIME := t#5s;
		POST_IGNITE_TIME :	TIME := t#25s;
		STAGE2_DELAY :	TIME := t#10s;
		SAFETY_TIME :	TIME := t#5s;
		LOCKOUT_TIME :	TIME := t#10s;
		MULTIPLE_IGNITION :	BOOL := TRUE;
		KW1 :	REAL;
		KW2 :	REAL;
		RUNTIME1 :	UDINT;
		RUNTIME2 :	UDINT;
		CYCLES :	UDINT;
		MOTOR :	BOOL;
		COIL1 :	BOOL;
		COIL2 :	BOOL;
		PRE_HEAT :	BOOL;
		IGNITE :	BOOL;
		KWH :	REAL;
		STATUS :	BYTE;
		FAIL :	BOOL;

		func_block : BURNER_Block;
	END_VAR
	func_block.IN := IN;
	func_block.STAGE2 := STAGE2;
	func_block.OVER_TEMP := OVER_TEMP ;
	func_block.OIL_TEMP    := OIL_TEMP    ;
	func_block.FLAME := FLAME;
	func_block.RST := RST;
	func_block.RST_TIMER := RST_TIMER ;
	func_block.PRE_HEAT_TIME := PRE_HEAT_TIME ;
	func_block.PRE_VENT_TIME    := PRE_VENT_TIME    ;
	func_block.PRE_IGNITE_TIME := PRE_IGNITE_TIME;
	func_block.POST_IGNITE_TIME := POST_IGNITE_TIME;
	func_block.STAGE2_DELAY := STAGE2_DELAY ;
	func_block.SAFETY_TIME := SAFETY_TIME ;
	func_block.LOCKOUT_TIME    := LOCKOUT_TIME    ;
	func_block.MULTIPLE_IGNITION := MULTIPLE_IGNITION;
	func_block.KW1 := KW1;
	func_block.KW2 := KW2;
	func_block.RUNTIME1 := RUNTIME1;
	func_block.RUNTIME2 := RUNTIME2;
	func_block.CYCLES := CYCLES;

	func_block();
	MOTOR  := func_block.MOTOR;
	COIL1  := func_block.COIL1;
	COIL2  := func_block.COIL2;
	PRE_HEAT  := func_block.PRE_HEAT;
	IGNITE  := func_block.IGNITE;
	KWH  := func_block.KWH;
	STATUS  := func_block.STATUS;
	FAIL  := func_block.FAIL;
	RUNTIME1  := func_block.RUNTIME1;
	RUNTIME2  := func_block.RUNTIME2;
	CYCLES  := func_block.CYCLES;
END_PROGRAM

CONFIGURATION Config0
	VAR_GLOBAL
		PLC_TICKS_PER_SEC :	INT;
		PLC_SYS_TICK_CNT :	DINT;
	END_VAR
  	RESOURCE Res0 ON PLC
    	TASK task0(INTERVAL := T#20ms,PRIORITY := 0);
    	PROGRAM instance0 WITH task0 : program0;
  	END_RESOURCE
END_CONFIGURATION

(* ---- lb_claude_assisted_5874272899fa_0006.st ---- *)
TYPE
  LOGLEVEL : (CRITICAL, WARNING, INFO, DEBUG) := INFO;
END_TYPE

FUNCTION_BLOCK LOGGER
  VAR_INPUT
    TRIG : BOOL;
    MSG : STRING;
    LEVEL : LOGLEVEL := INFO;
  END_VAR
  VAR
    TRIG0 : BOOL;
  END_VAR

  IF TRIG AND NOT TRIG0 THEN
  {{
   LogMessage(GetFbVar(LEVEL),(char*)GetFbVar(MSG, .body),GetFbVar(MSG, .len));
  }}
  END_IF;
  TRIG0:=TRIG;
END_FUNCTION_BLOCK

PROGRAM program0
  VAR
    I_PbFill : BOOL;
  END_VAR
  VAR
    Q_FillLight : BOOL;
  END_VAR
  VAR
    HMI_Fill : BOOL;
  END_VAR
  VAR
    Q_LightDischarge : BOOL;
  END_VAR
  VAR
    HMI_Dis : BOOL;
    Filling : BOOL;
    Discharging : BOOL;
    AutoMode : BOOL;
    Q_FillValve : INT;
    Q_DischargeValve : INT;
    Q_Display : INT;
    LevelRaw : INT;
    I_PbDischarge : BOOL;
  END_VAR
  VAR
    LevelPct : REAL;
    TimeFilling : TIME;
    TimeFillingInt : INT;
    TimeDiscarging : TIME;
    TimeDiscargingInt : INT;
    pbFill_prev : BOOL;
    pbDis_prev : BOOL;
    r_edge_fill : BOOL;
    r_edge_auto : BOOL;
    f_edge_dis : BOOL;
    PID0 : PID;
    AutoMode_prev : BOOL;
  END_VAR
  VAR
    SP : REAL := 30.0;
    PV : REAL;
    PV_lo : INT;
    PV_hi : INT;
    SP_lo : INT;
    SP_hi : INT;
  END_VAR
  VAR
    U_Manual : REAL;
    U_Auto : REAL;
  END_VAR
  VAR
    Kp : REAL := 4.0;
    Ki : REAL := 0.02;
    Kd : REAL := 0.4;
    Kp_lo : INT;
    Kp_hi : INT;
    Ki_lo : INT;
    Ki_hi : INT;
    Kd_lo : INT;
    Kd_hi : INT;
  END_VAR
  VAR
    tmp : REAL;
    IntTerm : REAL;
    Ts_s : REAL := 0.1;
    error : REAL;
    error_prev : REAL;
    derror : REAL;
    _raw_di : DINT;
    _loW : WORD;
    _hiW : WORD;
    _loDW : DWORD;
    _hiDW : DWORD;
    _raw_dw : DWORD;
  END_VAR

  _loDW   := WORD_TO_DWORD(INT_TO_WORD(Kp_lo));
  _hiDW   := SHL(WORD_TO_DWORD(INT_TO_WORD(Kp_hi)), 16);
  _raw_dw := _loDW OR _hiDW;
  _raw_di := DWORD_TO_DINT(_raw_dw);
  Kp := DINT_TO_REAL(_raw_di) / 10000.0;

  (* Repete para Ki/Kd *)
  _loDW   := WORD_TO_DWORD(INT_TO_WORD(Ki_lo));
  _hiDW   := SHL(WORD_TO_DWORD(INT_TO_WORD(Ki_hi)), 16);
  _raw_dw := _loDW OR _hiDW;
  _raw_di := DWORD_TO_DINT(_raw_dw);
  Ki := DINT_TO_REAL(_raw_di) / 10000.0;

  _loDW   := WORD_TO_DWORD(INT_TO_WORD(Kd_lo));
  _hiDW   := SHL(WORD_TO_DWORD(INT_TO_WORD(Kd_hi)), 16);
  _raw_dw := _loDW OR _hiDW;
  _raw_di := DWORD_TO_DINT(_raw_dw);
  Kd := DINT_TO_REAL(_raw_di) / 10000.0;

  _loDW   := WORD_TO_DWORD(INT_TO_WORD(SP_lo));
  _hiDW   := SHL(WORD_TO_DWORD(INT_TO_WORD(SP_hi)), 16);
  _raw_dw := _loDW OR _hiDW;
  _raw_di := DWORD_TO_DINT(_raw_dw);
  SP := DINT_TO_REAL(_raw_di) / 10000.0;

  (* PV já está em 0..1 (ex.: calculado de LevelRaw). Agora exporta em LO/HI ×10000 *)
  _raw_di := REAL_TO_DINT(PV * 10000.0);
  _raw_dw := DINT_TO_DWORD(_raw_di);

  PV_lo := WORD_TO_INT(DWORD_TO_WORD(_raw_dw));                 (* LOW  *)
  PV_hi := WORD_TO_INT(DWORD_TO_WORD(SHR(_raw_dw, 16)));        (* HIGH *)

      (* ===== Factory IO Inputs ===== *)

      r_edge_fill := I_PbFill AND NOT pbFill_prev;

      f_edge_dis  := pbDis_prev AND NOT I_PbDischarge;

      pbFill_prev := I_PbFill;

      pbDis_prev  := I_PbDischarge;

      IF r_edge_fill AND NOT Discharging AND NOT AutoMode THEN

          Filling := TRUE;

          (* reset PID ao iniciar *)

          IntTerm    := 0.0;

          error_prev := 0.0;

      END_IF;

      IF f_edge_dis AND NOT AutoMode THEN

          Discharging := TRUE;

          Filling     := FALSE;

          (* reset geral ao descarregar *)

          IntTerm    := 0.0;

          error_prev := 0.0;

      END_IF;

      (* ======= PV =======  (0..1) *)

      tmp := INT_TO_REAL(LevelRaw) / 1000.0;

      IF tmp < 0.0 THEN tmp := 0.0; END_IF;

      IF tmp > 1.0 THEN tmp := 1.0; END_IF;

      LevelPct := tmp * 100.0;    (* 0..100 *)

      PV       := tmp;            (* 0..1 *)

      (* auto stop da descarga quando ~0% *)

      IF Discharging AND ((PV * 100.0) <= 1.0) THEN

          Discharging := FALSE;

      END_IF;

      (* ======= AUTO/MAN MODE =======  *)

      r_edge_auto := AutoMode AND NOT AutoMode_prev;

      AutoMode_prev := AutoMode;

      IF AutoMode THEN

          (* reset só quando entra em AUTO *)

          IF r_edge_auto THEN

              Filling     := FALSE;

              Discharging := FALSE;

              IntTerm     := 0.0;

              error_prev  := 0.0;

              U_Auto      := 0.0;

          END_IF;

          (* ---------- PID SEMPRE ATIVO NO AUTO ---------- *)

          error   := (SP / 100.0) - PV;

          IntTerm := IntTerm + (Ki * error * Ts_s);

          derror  := (error - error_prev) / Ts_s;

          U_Auto := (Kp * error) + IntTerm + (Kd * derror);

          (* saturação *)

          IF U_Auto >  1.0 THEN U_Auto :=  1.0; END_IF;

          IF U_Auto < -1.0 THEN U_Auto := -1.0; END_IF;

          (* anti-windup *)

          IF ((U_Auto =  1.0) AND (error > 0.0)) OR

             ((U_Auto = -1.0) AND (error < 0.0)) THEN

              IntTerm := IntTerm - (Ki * error * Ts_s);

          END_IF;

          (* mapeamento 0..1000 e estados *)

          IF U_Auto > 0.0 THEN

              Q_FillValve      := REAL_TO_INT(1000.0 *  U_Auto);

              Q_DischargeValve := 0;

              Filling          := TRUE;

              Discharging      := FALSE;

          ELSIF U_Auto < 0.0 THEN

              Q_DischargeValve := REAL_TO_INT(1000.0 * (-U_Auto));

              Q_FillValve      := 0;

              Filling          := FALSE;

              Discharging      := TRUE;

          ELSE

              Q_FillValve      := 0;

              Q_DischargeValve := 0;

              Filling          := FALSE;

              Discharging      := FALSE;

          END_IF;

      (* ---------- MANUAL ---------- *)

      ELSE

          IF HMI_Dis THEN

              Q_DischargeValve := 1000;

              Q_FillValve      := 0;

              Discharging      := TRUE;

              Filling          := FALSE;

          ELSIF HMI_Fill THEN

              Q_FillValve      := 1000;   (* abre 100% *)

              Q_DischargeValve := 0;

              Filling          := TRUE;

              Discharging      := FALSE;

          ELSE

              HMI_Dis          := 0;

              Q_FillValve      := 0;

              Q_DischargeValve := 0;

              Filling          := FALSE;

              Discharging      := FALSE;

          END_IF;

      END_IF;

      error            := (SP / 100.0) - PV;

      error_prev       := error;

      Q_Display        := REAL_TO_INT(PV * 100.0);

      Q_FillLight      := Filling;

      Q_LightDischarge := Discharging;
END_PROGRAM

CONFIGURATION Config0

  RESOURCE Res0 ON PLC
    TASK task0(INTERVAL := T#20ms,PRIORITY := 0);
    PROGRAM instance0 WITH task0 : program0;
  END_RESOURCE
END_CONFIGURATION

(* ---- lb_claude_assisted_5a229da37ffe_0002.st ---- *)
FUNCTION_BLOCK T_PLC_MS_block
	VAR_OUTPUT
		T_PLC_MS :	UDINT;
	END_VAR

	VAR
		PLC_TICKS_PER_SEC :	INT;
		PLC_SYS_TICK_CNT :	DINT;
	END_VAR

	VAR
		debug :	BOOL;(*Debug-Mode ON / OFF*)
		N :	INT;(*Debug-Faktor*)
		Offset :	UDINT;(*Debug-Offset*)
		temp :	DWORD := DWORD#1;(*Debug-Offset*)
		MODE :	BOOL;(*modus*)
		faktor :	UDINT;(*Systemtakt-Faktor*)
		init :	BOOL;
		v_plc_ticks_per_sec :	UDINT;
		base :	UDINT := UDINT#1000;
	END_VAR

	IF init = FALSE THEN
		v_plc_ticks_per_sec := INT_TO_UDINT(PLC_TICKS_PER_SEC);
		IF v_plc_ticks_per_sec = UDINT#1024 THEN
			faktor := UDINT#1;
			MODE := FALSE;
		ELSIF v_plc_ticks_per_sec > UDINT#0 THEN
			IF v_plc_ticks_per_sec <= base THEN
				faktor := base / v_plc_ticks_per_sec;
				MODE := FALSE;
			ELSE
				faktor := v_plc_ticks_per_sec / base;
				MODE := TRUE;
			END_IF;
		ELSE
			faktor := UDINT#1;
		END_IF;
		init := TRUE;
	END_IF;

	IF MODE THEN
		T_PLC_MS := DINT_TO_UDINT(PLC_SYS_TICK_CNT) / faktor;
	ELSE
		T_PLC_MS := DINT_TO_UDINT(PLC_SYS_TICK_CNT) * faktor;
	END_IF;

	IF debug THEN
		T_PLC_MS := (DWORD_TO_UDINT(SHL(UDINT_TO_DWORD(T_PLC_MS),N) OR SHL(temp,N)) - UDINT#1) + Offset;
	END_IF;
END_FUNCTION_BLOCK

FUNCTION TIME_TO_UDINT2:UDINT
	VAR_INPUT
		X :	TIME;
	END_VAR

	TIME_TO_UDINT2 := DINT_TO_UDINT(TIME_TO_DINT(X));
END_FUNCTION

FUNCTION_BLOCK TUNE_Block

	VAR_INPUT
		SET :	BOOL;
		SU :	BOOL;
		SD :	BOOL;
		RST :	BOOL;
		SS :	REAL := 0.1;
		LIMIT_L :	REAL;
		LIMIT_H :	REAL := 100.0;
		RST_VAL :	REAL;
		SET_VAL :	REAL := 100.0;
		T1 :	TIME := T#500ms;
		T2 :	TIME := T#2s;
		S1 :	REAL := 2.0;
		S2 :	REAL := 10.0;
	END_VAR

	VAR_OUTPUT
		Y :	REAL;
	END_VAR

	VAR
		TX :	UDINT;
		START :	UDINT;
		START2 :	UDINT;
		STATE :	INT;
		IN :	BOOL;
		STEP2 :	REAL;
		SPEED :	REAL;
		Y_START :	REAL;
		Y_START2 :	REAL;
		T_PLC_MS :	T_PLC_MS_block;
	END_VAR

	T_PLC_MS();
	TX:= T_PLC_MS.T_PLC_MS;

	IF RST THEN
		Y := RST_VAL;
		STATE := 0;
	ELSIF SET THEN
		Y := SET_VAL;
		STATE := 0;
	ELSIF STATE > 0 THEN
		IF STATE = 1 THEN
			IN := su;
		ELSE
			IN := sd;
		END_IF;
		IF NOT IN AND TX - START <= TIME_TO_UDINT2(T1) THEN
			Y := Y_START + STEP2;
			STATE := 0;
		ELSIF IN AND TX - START >= TIME_TO_UDINT2(T2) THEN
			Y := Y_START2 + UDINT_TO_REAL(TX - START2) * S2 / SPEED;
		ELSIF IN AND TX - START >= TIME_TO_UDINT2(T1) THEN
			Y := Y_START + UDINT_TO_REAL(TX - START - TIME_TO_UDINT2(T1)) * S1 / SPEED;
			START2 := TX;
			Y_START2 := Y;
		ELSIF NOT IN THEN
			STATE := 0;
		END_IF;
	ELSIF su THEN
		STATE := 1;
		START := TX;
		STEP2 := ss;
		SPEED := 1000.0;
		Y_START := Y;
	ELSIF sd THEN

		STATE := 2;
		START := TX;
		STEP2 := -ss;
		SPEED := -1000.0;
		Y_START := Y;
	END_IF;

END_FUNCTION_BLOCK

PROGRAM program0
  	VAR
		SET :	BOOL;
		SU :	BOOL;
		SD :	BOOL;
		RST :	BOOL;
		SS :	REAL := 0.1;
		LIMIT_L :	REAL;
		LIMIT_H :	REAL := 100.0;
		RST_VAL :	REAL;
		SET_VAL :	REAL := 100.0;
		T1 :	TIME := T#500ms;
		T2 :	TIME := T#2s;
		S1 :	REAL := 2.0;
		S2 :	REAL := 10.0;
		Y :	REAL;
		func_block : TUNE_Block;
  	END_VAR
	func_block.SET := SET;
	func_block.SU := SU;
	func_block.SD := SD;
	func_block.RST := RST;
	func_block.SS:= SS;
	func_block.LIMIT_L := LIMIT_L;
	func_block.LIMIT_H := LIMIT_H;
	func_block.RST_VAL := RST_VAL;
	func_block.SET_VAL := SET_VAL;
	func_block.T1 := T1;
	func_block.T2 := T2;
	func_block.S1 := S1;
	func_block.S2 := S2;
	func_block();
	Y := func_block.Y;
END_PROGRAM

(* ---- lb_claude_assisted_5b1ea319f143_0119.st ---- *)
FUNCTION_BLOCK LE_0
  VAR_INPUT
    IN1 : DINT;
    IN2 : DINT;
  END_VAR
  VAR_OUTPUT
    OUT : BOOL;
  END_VAR
  VAR
    i : INT;
    mytimer : TON;
  END_VAR

  OUT:=FALSE;
  IF IN1<=IN2 then
    OUT:=TRUE;
  END_IF;
  mytimer(IN := TRUE, PT := t#8000ms);
  i:=0;
  IF mytimer.Q = TRUE then
     WHILE i<4 do
      OUT:=TRUE;
    End_WHILE;
  End_IF;
END_FUNCTION_BLOCK

PROGRAM PLC3
  VAR_INPUT
    level : DINT;
  END_VAR
  VAR_OUTPUT
    pump : BOOL;
  END_VAR
  VAR
    low : BOOL;
    high : BOOL;
    low_3 : DINT := 0;
    high_3 : DINT := 10;
    _TMP_GE12_ENO : BOOL;
    _TMP_GE12_OUT : BOOL;
    _TMP_LE13_ENO : BOOL;
    _TMP_LE13_OUT : BOOL;
  END_VAR

  _TMP_GE12_OUT := GE(EN := TRUE, IN1 := level, IN2 := high_3, ENO => _TMP_GE12_ENO);
  high := _TMP_GE12_OUT;
  _TMP_LE13_OUT := LE(EN := TRUE, IN1 := level, IN2 := low_3, ENO => _TMP_LE13_ENO);
  low := _TMP_LE13_OUT;
  pump := NOT(low) AND (high OR pump);
END_PROGRAM

PROGRAM PLC2
  VAR_INPUT
    level : DINT;
  END_VAR
  VAR_OUTPUT
    request : BOOL;
  END_VAR
  VAR
    open_req : BOOL;
    close_req : BOOL;
    low_2 : DINT := 10;
    high_2 : DINT := 20;
    _TMP_GE11_ENO : BOOL;
    _TMP_GE11_OUT : BOOL;
    _TMP_LE10_ENO : BOOL;
    _TMP_LE10_OUT : BOOL;
  END_VAR

  _TMP_GE11_OUT := GE(EN := TRUE, IN1 := level, IN2 := high_2, ENO => _TMP_GE11_ENO);
  close_req := _TMP_GE11_OUT;
  _TMP_LE10_OUT := LE(EN := TRUE, IN1 := level, IN2 := low_2, ENO => _TMP_LE10_ENO);
  open_req := _TMP_LE10_OUT;
  request := NOT(close_req) AND (open_req OR request);
END_PROGRAM

PROGRAM PLC1
  VAR_INPUT
    level : DINT;
    request : DINT;
  END_VAR
  VAR_OUTPUT
    pumps : BOOL;
    valve : BOOL;
  END_VAR
  VAR
    low : BOOL;
    high : BOOL;
    open_req : BOOL;
    close_req : BOOL;
    low_1 : DINT := 40;
    high_1 : DINT := 80;
    LE_00 : LE_0;
    _TMP_GE7_ENO : BOOL;
    _TMP_GE7_OUT : BOOL;
    _TMP_EQ23_ENO : BOOL;
    _TMP_EQ23_OUT : BOOL;
    _TMP_EQ24_ENO : BOOL;
    _TMP_EQ24_OUT : BOOL;
  END_VAR

  _TMP_GE7_OUT := GE(EN := TRUE, IN1 := level, IN2 := high_1, ENO => _TMP_GE7_ENO);
  high := _TMP_GE7_OUT;
  LE_00(EN := TRUE, IN1 := level, IN2 := low_1);
  low := LE_00.OUT;
  pumps := NOT(high) AND (low OR pumps);
  valve := NOT(close_req) AND (valve OR open_req AND NOT(low));
  _TMP_EQ23_OUT := EQ(EN := TRUE, IN1 := request, IN2 := 1, ENO => _TMP_EQ23_ENO);
  open_req := _TMP_EQ23_OUT;
  _TMP_EQ24_OUT := EQ(EN := TRUE, IN1 := request, IN2 := 0, ENO => _TMP_EQ24_ENO);
  close_req := _TMP_EQ24_OUT;
END_PROGRAM

CONFIGURATION Config0

  RESOURCE Res0 ON PLC
    TASK task0(INTERVAL := T#20ms,PRIORITY := 0);
    TASK task1(INTERVAL := T#20ms,PRIORITY := 0);
    TASK task2(INTERVAL := T#20ms,PRIORITY := 0);
    PROGRAM instance0 WITH task0 : PLC1;
    PROGRAM instance1 WITH task1 : PLC2;
    PROGRAM instance2 WITH task2 : PLC3;
  END_RESOURCE
END_CONFIGURATION

(* ---- lb_claude_assisted_5b42ddb50301_0036.st ---- *)
(*
This code implements a randomly grown symbolic expression:

!((IN16 & IN32) & ((xor(xor(xor(xor(IN24 | IN48, (((xor(xor(xor(xor(IN40, true), IN7), xor(xor(IN27, IN44), IN7)), IN6 | IN4)) & ((IN19 | IN14) & (IN40 & IN35))) & ((xor(xor(xor(xor(IN39, IN34), IN48), IN14), IN40)) | ((xor(xor(IN13, IN28), IN42)) & IN45))) & (!(((IN21 | IN2) & (xor(xor(IN10, IN37), IN37))) & (!(IN11))))), xor(xor(xor(xor(xor(xor(IN7, IN46), !(!(IN6))), !(!(IN40 & IN29))), ((IN46 | IN37) & IN8) & ((IN22 | IN10) & (!(IN45)))), IN18 & (((IN3 & IN7) | IN33) | (xor(xor(!(IN41), IN45), IN34 | IN4)))), (xor(xor(xor(xor(!(IN48), true), IN37), IN21), xor(xor(xor(xor(IN22, IN49), IN18), IN23 & IN36), xor(xor(IN50, IN46), IN46)))) & (!((IN47 & IN2) | (IN33 | IN12))))), !(IN49 | ((((!(IN38)) | (IN39 | IN16)) & ((IN6 | IN42) | IN24)) & (!((!(IN17)) & (true | IN18)))))), IN1)) & ((xor(xor(IN37, xor(xor(!(((IN10 | IN47) & (xor(xor(IN39, IN25), IN32))) & (xor(xor(!(IN11), IN27 | IN31), xor(xor(IN28, IN4), IN40)))), (xor(xor(!(IN50 & IN31), IN44), !(IN17 & IN29))) & ((!(IN47)) | ((!(IN16)) & (!(IN24))))), xor(xor(((!(IN19)) & (xor(xor(IN38, IN13), false))) & (xor(xor(IN15, IN34 | IN14), !(IN33))), xor(xor((xor(xor(IN39, IN24), IN44)) & IN42, (!(IN24)) & (xor(xor(IN23, IN12), IN20))), (xor(xor(false, IN3), IN48)) | (xor(xor(IN8, IN18), IN19)))), !((!(IN28)) | IN33)))), xor(xor(!(!(!(IN26 & false))), IN33), IN30 | ((IN48 | IN35) & (xor(xor(IN11 & IN12, IN29 | IN41), !(IN30))))))) & (xor(xor((IN8 & (!((IN8 | IN46) & IN22))) & (((!(IN29 & IN32)) | ((IN9 | IN45) & (!(IN24)))) | (((!(IN41)) | (xor(xor(IN1, IN37), IN29))) & ((IN13 | IN50) | (IN37 | IN11)))), !((xor(xor((IN17 | IN14) | (xor(xor(IN15, true), IN25)), !(xor(xor(IN2, IN26), IN23))), (IN37 | IN15) | (IN44 | IN22))) | ((xor(xor(xor(xor(IN23, IN31), IN33), IN39 | IN21), IN21)) | (!(!(IN19)))))), (!(((IN24 | false) | (xor(xor(IN17, IN50), IN9))) | (xor(xor(IN39 & IN35, IN19 & IN48), IN37 & IN25)))) | IN46)))))

*)

FUNCTION_BLOCK F_CollectInput
  VAR_IN_OUT
      Data : ARRAY[1..50] OF BOOL;
  END_VAR
  VAR_INPUT
      TICK  : BOOL := 0;
      IN1   : BOOL := 0;
      IN2   : BOOL := 0;
      IN3   : BOOL := 0;
      IN4   : BOOL := 0;
      IN5   : BOOL := 0;
      RESET : BOOL := FALSE;
  END_VAR
  VAR_OUTPUT
      Finished : BOOL;
  END_VAR
  VAR
      j    : USINT := 1;
      tock : BOOL  := 0;
  END_VAR
  IF NOT RESET AND tock = NOT TICK THEN
      Data[j]   := IN1;
      Data[j+1] := IN2;
      Data[j+2] := IN3;
      Data[j+3] := IN4;
      Data[j+4] := IN5;
      j := j + 5;
      tock := TICK;
  ELSE
      j := 1;
      tock := 0;
  END_IF;
  Finished := (j > 50);
END_FUNCTION_BLOCK

PROGRAM Boiler
  VAR
    Data  : ARRAY[1..50] OF BOOL;
    Ready : BOOL;
    CollectInput : F_CollectInput;
  END_VAR
  VAR
    TICK     AT %IX1.0 : BOOL;
    IN1      AT %IX0.3 : BOOL;
    IN2      AT %IX0.4 : BOOL;
    IN3      AT %IX0.5 : BOOL;
    IN4      AT %IX0.6 : BOOL;
    IN5      AT %IX0.7 : BOOL;
    OutReady AT %QX0.0 : BOOL := FALSE;
    FeedNext AT %QX0.1 : BOOL := FALSE;
    Out      AT %QX0.2 : BOOL;
  END_VAR
  CollectInput(TICK:=TICK, IN1:=IN1, IN2:=IN2, IN3:=IN3, IN4:=IN4, IN5:=IN5);
  Ready := CollectInput.Finished;
  FeedNext := 1;
  IF Ready THEN
    Out := (NOT ((Data[16] AND Data[32]) AND ((((((Data[24] OR Data[48]) XOR (((((((Data[40] XOR TRUE) XOR Data[7]) XOR ((Data[27] XOR Data[44]) XOR Data[7])) XOR (Data[6] OR Data[4])) AND ((Data[19] OR Data[14]) AND (Data[40] AND Data[35]))) AND (((((Data[39] XOR Data[34]) XOR Data[48]) XOR Data[14]) XOR Data[40]) OR (((Data[13] XOR Data[28]) XOR Data[42]) AND Data[45]))) AND (NOT (((Data[21] OR Data[2]) AND ((Data[10] XOR Data[37]) XOR Data[37])) AND (NOT Data[11]))))) XOR ((((((Data[7] XOR Data[46]) XOR (NOT (NOT Data[6]))) XOR (NOT (NOT (Data[40] AND Data[29])))) XOR (((Data[46] OR Data[37]) AND Data[8]) AND ((Data[22] OR Data[10]) AND (NOT Data[45])))) XOR (Data[18] AND (((Data[3] AND Data[7]) OR Data[33]) OR (((NOT Data[41]) XOR Data[45]) XOR (Data[34] OR Data[4]))))) XOR ((((((NOT Data[48]) XOR TRUE) XOR Data[37]) XOR Data[21]) XOR ((((Data[22] XOR Data[49]) XOR Data[18]) XOR (Data[23] AND Data[36])) XOR ((Data[50] XOR Data[46]) XOR Data[46]))) AND (NOT ((Data[47] AND Data[2]) OR (Data[33] OR Data[12])))))) XOR (NOT (Data[49] OR ((((NOT Data[38]) OR (Data[39] OR Data[16])) AND ((Data[6] OR Data[42]) OR Data[24])) AND (NOT ((NOT Data[17]) AND (TRUE OR Data[18]))))))) XOR Data[1]) AND (((Data[37] XOR (((NOT (((Data[10] OR Data[47]) AND ((Data[39] XOR Data[25]) XOR Data[32])) AND (((NOT Data[11]) XOR (Data[27] OR Data[31])) XOR ((Data[28] XOR Data[4]) XOR Data[40])))) XOR ((((NOT (Data[50] AND Data[31])) XOR Data[44]) XOR (NOT (Data[17] AND Data[29]))) AND ((NOT Data[47]) OR ((NOT Data[16]) AND (NOT Data[24]))))) XOR (((((NOT Data[19]) AND ((Data[38] XOR Data[13]) XOR FALSE)) AND ((Data[15] XOR (Data[34] OR Data[14])) XOR (NOT Data[33]))) XOR (((((Data[39] XOR Data[24]) XOR Data[44]) AND Data[42]) XOR ((NOT Data[24]) AND ((Data[23] XOR Data[12]) XOR Data[20]))) XOR (((FALSE XOR Data[3]) XOR Data[48]) OR ((Data[8] XOR Data[18]) XOR Data[19])))) XOR (NOT ((NOT Data[28]) OR Data[33]))))) XOR (((NOT (NOT (NOT (Data[26] AND FALSE)))) XOR Data[33]) XOR (Data[30] OR ((Data[48] OR Data[35]) AND (((Data[11] AND Data[12]) XOR (Data[29] OR Data[41])) XOR (NOT Data[30])))))) AND ((((Data[8] AND (NOT ((Data[8] OR Data[46]) AND Data[22]))) AND (((NOT (Data[29] AND Data[32])) OR ((Data[9] OR Data[45]) AND (NOT Data[24]))) OR (((NOT Data[41]) OR ((Data[1] XOR Data[37]) XOR Data[29])) AND ((Data[13] OR Data[50]) OR (Data[37] OR Data[11]))))) XOR (NOT (((((Data[17] OR Data[14]) OR ((Data[15] XOR TRUE) XOR Data[25])) XOR (NOT ((Data[2] XOR Data[26]) XOR Data[23]))) XOR ((Data[37] OR Data[15]) OR (Data[44] OR Data[22]))) OR (((((Data[23] XOR Data[31]) XOR Data[33]) XOR (Data[39] OR Data[21])) XOR Data[21]) OR (NOT (NOT Data[19])))))) XOR ((NOT (((Data[24] OR FALSE) OR ((Data[17] XOR Data[50]) XOR Data[9])) OR (((Data[39] AND Data[35]) XOR (Data[19] AND Data[48])) XOR (Data[37] AND Data[25])))) OR Data[46]))))));
    OutReady := 1;
    CollectInput(RESET:=TRUE);
  END_IF;
END_PROGRAM

CONFIGURATION Config0
  RESOURCE Res0 ON PLC
    TASK task0(INTERVAL := T#20ms,PRIORITY := 0);
    PROGRAM instance0 WITH task0 : Boiler;
  END_RESOURCE
END_CONFIGURATION
